(* IEC 61131-3 sources: Advanced_PLCs_Midterm_Project/Source_Code/Advanced_Midterm_PLC_Code/Dan_Thermostat_Code/Thermo_Code, 1 file *)

(* ---- HMI.plc ---- *)
PROGRAM PageDraw WITH Draw;
PROGRAM PageRefresh WITH Refresh;

	(***************************)
	(*                         *)
	(*     GLOBAL VARIABLES    *)
	(*                         *)
	(***************************)

VAR_GLOBAL

	{G:"Call stack"}
	giStackPtr : INT := -1;
	guiCallStack : ARRAY[ 0..9 ] OF UINT;

	{G:"Back buffer"}
	$giBackBufferCurr : INT := -1;
	$giBackBufferFirst : INT := -1;
	$giBackBufferLast : INT := -1;
	$guiBackBuffer : ARRAY[ 0..9 ] OF UINT;

	{G:"Sets"}
	$PagIndex : UINT;
	$PagNumber : UINT;
	$waitRefresh : BOOL;

	{G:"page1_vars"}
	fbpage1 : Drawpage1;
	fbRefrpage1 : Refrpage1;
	fbpage1String_1 : Static02 := (x:=58, y:=75, pFont:=?EWP2_8x16, bckCol:=12632256, pString:=?kStr00001, pVisVar:=1, format:=16#0020, bordPts:=0, selForeCol:=12632256, pRefrVar:=0, pSelVar:=0, numChars:=0);
	fbpage1String_4 : Static02 := (wHnd:=1, x:=54, y:=156, pFont:=?EWP2_8x16, bckCol:=12632256, pString:=?kStr00002, pVisVar:=1, format:=16#0020, bordPts:=0, selForeCol:=12632256, pRefrVar:=0, pSelVar:=0, numChars:=0);
	fbpage1Edit_3 : EditBox03 := (wHnd:=2, x1:=94, y1:=186, x2:=157, y2:=201, pFont:=?EWP2_8x16, bckCol:=32767, bordPts:=1, rw:=TRUE, pVar:=16#00201100, order:=2, pVisVar:=1, foreSelCol:=12632256, refr:=TRUE, type:=tyInt, format:=16#2100000C, pCanSel:=1, pEnumId:=0);
	fbpage1Edit_5 : EditBox03 := (wHnd:=3, x1:=91, y1:=100, x2:=154, y2:=115, pFont:=?EWP2_8x16, bckCol:=65535, bordPts:=1, rw:=TRUE, pVar:=16#00201000, order:=3, pVisVar:=1, foreSelCol:=12632256, refr:=TRUE, type:=tyInt, format:=16#2100000C, pCanSel:=1, pEnumId:=0);

	{G:"Back page manager"}
	fbBackPage : DrawBackPage;

END_VAR

	(***************************)
	(*                         *)
	(*        CONSTANTS        *)
	(*                         *)
	(***************************)

VAR_GLOBAL CONSTANT

	kStr00002 :STRING[18] := 'Relative Humidity';
	kStr00001 :STRING[19] := 'Temperature[deg F]';

END_VAR
VAR_GLOBAL CONSTANT

	{G:"Fonts"}
	EWP2_8x16_len : USINT := 8;
	EWP2_8x16_hei : USINT := 16;
	EWP2_8x16_offs : USINT := 0;
	EWP2_8x16 AT %MB1000.0 : ARRAY[ 0..2095 ] OF BYTE := 254,8,16,0,95,2,0,32,0,33,0,34,0,35,0,36,
				0,37,0,38,0,39,0,40,0,41,0,42,0,43,0,44,
				0,45,0,46,0,47,0,48,0,49,0,50,0,51,0,52,
				0,53,0,54,0,55,0,56,0,57,0,58,0,59,0,60,
				0,61,0,62,0,63,0,64,0,65,0,66,0,67,0,68,
				0,69,0,70,0,71,0,72,0,73,0,74,0,75,0,76,
				0,77,0,78,0,79,0,80,0,81,0,82,0,83,0,84,
				0,85,0,86,0,87,0,88,0,89,0,90,0,91,0,92,
				0,93,0,94,0,95,0,96,0,97,0,98,0,99,0,100,
				0,101,0,102,0,103,0,104,0,105,0,106,0,107,0,108,
				0,109,0,110,0,111,0,112,0,113,0,114,0,115,0,116,
				0,117,0,118,0,119,0,120,0,121,0,122,0,123,0,124,
				0,125,0,126,7(0),16,3(0),32,3(0),48,3(0),64,3(0),80,3(0),96,
				3(0),112,3(0),128,3(0),144,3(0),160,3(0),176,3(0),192,3(0),208,3(0),224,
				3(0),240,0,0,1,3(0),1,16,0,0,1,32,0,0,1,48,
				0,0,1,64,0,0,1,80,0,0,1,96,0,0,1,112,
				0,0,1,128,0,0,1,144,0,0,1,160,0,0,1,176,
				0,0,1,192,0,0,1,208,0,0,1,224,0,0,1,240,
				0,0,2,3(0),2,16,0,0,2,32,0,0,2,48,0,0,
				2,64,0,0,2,80,0,0,2,96,0,0,2,112,0,0,
				2,128,0,0,2,144,0,0,2,160,0,0,2,176,0,0,
				2,192,0,0,2,208,0,0,2,224,0,0,2,240,0,0,
				3,3(0),3,16,0,0,3,32,0,0,3,48,0,0,3,64,
				0,0,3,80,0,0,3,96,0,0,3,112,0,0,3,128,
				0,0,3,144,0,0,3,160,0,0,3,176,0,0,3,192,
				0,0,3,208,0,0,3,224,0,0,3,240,0,0,4,3(0),
				4,16,0,0,4,32,0,0,4,48,0,0,4,64,0,0,
				4,80,0,0,4,96,0,0,4,112,0,0,4,128,0,0,
				4,144,0,0,4,160,0,0,4,176,0,0,4,192,0,0,
				4,208,0,0,4,224,0,0,4,240,0,0,5,3(0),5,16,
				0,0,5,32,0,0,5,48,0,0,5,64,0,0,5,80,
				0,0,5,96,0,0,5,112,0,0,5,128,0,0,5,144,
				0,0,5,160,0,0,5,176,0,0,5,192,0,0,5,208,
				0,0,5,224,19(0),252,252,6(0),13,13,5(0),60,60,0,60,60,
				9(0),32,32,224,252,60,224,252,60,1,15,15,1,15,15,1,
				1,0,0,56,124,254,254,132,4,0,0,8,8,31,31,15,
				7,56,124,68,252,248,248,156,132,0,8,14,7,7,15,8,
				15,0,0,184,252,228,188,152,192,0,7,15,8,9,15,7,
				13,3(0),60,60,14(0),192,240,56,12,4,3(0),3,15,28,48,32,
				0,4,12,56,240,192,3(0),32,48,28,15,3,3(0),40,56,124,
				124,56,40,10(0),3(128),240,240,128,128,4(0),7,7,12(0),16,28,12,
				13(0),5(1),12(0),12,12,6(0),192,240,60,12,0,0,12,15,3,5(0),
				240,248,204,196,204,248,240,0,3,7,12,8,12,7,3,0,
				8,12,252,252,4(0),8,8,15,15,8,8,0,0,3(4),132,252,
				120,0,0,12,14,11,9,8,8,0,0,4,68,68,228,188,
				24,0,0,3(8),12,7,3,3(0),192,240,60,252,252,0,0,3,
				3,2,2,15,15,2,0,0,124,124,68,68,196,132,0,0,
				4(8),15,7,0,240,248,204,68,68,196,128,0,3,7,12,8,
				8,15,7,0,3(4),196,244,60,12,0,0,8,14,7,1,3(0),
				24,188,228,68,228,188,24,0,7,15,3(8),15,7,0,120,252,
				132,132,204,248,240,0,0,3(8),12,7,3,3(0),96,96,6(0),12,
				12,6(0),96,96,5(0),16,28,12,5(0),128,192,64,96,48,16,3(0),
				1,1,3,6,4,0,7(32),0,7(1),0,0,16,48,96,64,192,
				128,0,0,4,6,3,1,1,3(0),8,140,196,68,124,56,3(0),
				13,13,3(0),240,248,204,228,228,236,248,240,7,15,25,4(19),1,
				0,128,248,124,124,248,128,0,12,15,3,1,1,3,15,12,
				0,252,252,3(68),252,184,0,15,15,3(8),15,7,0,240,248,12,
				4,4,12,8,0,3,7,12,8,8,12,4,0,252,252,4,
				4,12,248,240,0,15,15,8,8,12,7,3,0,252,252,5(68),
				0,15,15,5(8),0,252,252,5(68),0,15,15,6(0),240,248,12,132,
				132,140,136,0,3,7,12,8,8,15,7,0,252,252,3(64),252,
				252,0,15,15,3(0),15,15,0,4,4,252,252,4,4,0,0,
				8,8,15,15,8,8,6(0),252,252,0,0,4(8),15,7,0,0,
				252,252,192,224,48,24,12,0,15,15,0,1,3,6,12,0,
				252,252,6(0),15,15,5(8),0,252,252,120,96,120,252,252,0,15,
				15,3(0),15,15,0,252,252,120,224,128,252,252,0,15,15,0,
				1,7,15,15,0,240,248,12,4,12,248,240,0,3,7,12,
				8,12,7,3,0,252,252,3(68),124,56,0,15,15,6(0),240,248,
				12,4,12,248,240,0,3,7,12,24,60,39,35,0,252,252,
				68,196,196,124,56,0,15,15,0,0,3,7,12,0,56,124,
				68,196,132,140,8,0,4,12,3(8),15,7,3(4),252,252,3(4),3(0),
				15,15,4(0),252,252,3(0),252,252,0,7,15,3(8),15,7,12,124,
				240,128,128,240,124,12,0,0,7,15,15,7,0,0,252,252,
				128,224,224,128,252,252,3,15,15,3,3,15,15,3,4,28,
				56,224,224,56,28,4,8,14,7,1,1,7,14,8,4,28,
				56,224,224,56,28,4,3(0),15,15,4(0),4,4,132,228,116,28,
				12,0,12,14,11,9,3(8),3(0),252,252,4,4,4(0),63,63,32,
				32,0,0,12,60,240,192,7(0),3,15,12,0,0,4,4,252,
				252,4(0),32,32,63,63,4(0),64,112,56,12,12,56,112,16(0),8(64),
				3(0),4,12,8,11(0),64,96,3(32),224,192,0,6,15,9,9,13,
				15,15,0,252,252,96,32,96,192,128,0,15,15,12,8,12,
				7,3,0,128,192,96,4(32),0,3,7,12,4(8),0,128,192,96,
				32,96,252,252,0,3,7,12,8,12,15,15,0,128,192,96,
				32,96,192,128,0,3,7,13,4(9),0,32,32,248,252,3(36),3(0),
				15,15,4(0),192,224,32,32,224,224,32,0,61,127,74,74,75,
				121,48,0,252,252,96,32,32,224,192,0,15,15,3(0),15,15,
				0,0,32,32,228,228,6(0),15,15,4(0),32,32,228,228,3(0),3(64),
				127,63,3(0),252,252,128,192,96,32,0,0,15,15,1,3,6,
				12,8,0,4,4,252,252,6(0),15,15,8,8,0,224,224,32,
				224,224,32,224,192,15,15,0,15,15,0,15,15,0,224,224,
				96,32,32,224,192,0,15,15,3(0),15,15,0,192,224,3(32),224,
				192,0,7,15,3(8),15,7,0,224,224,96,32,96,192,128,0,
				127,127,12,8,12,7,3,0,128,192,96,32,96,224,224,0,
				3,7,12,8,12,127,127,0,0,224,224,96,3(32),0,0,15,
				15,5(0),192,224,5(32),0,8,4(9),15,6,0,0,32,248,248,32,
				32,4(0),7,15,3(8),0,224,224,3(0),224,224,0,7,15,8,8,
				12,15,15,32,224,192,0,0,192,224,32,0,1,7,14,14,
				7,1,0,224,224,0,128,128,0,224,224,3,15,15,3,3,
				15,15,3,0,32,96,192,128,192,96,32,0,8,12,7,3,
				7,12,8,32,224,192,0,0,192,224,32,64,64,103,63,31,
				7,3(0),3(32),160,224,96,32,0,8,12,15,11,3(8),0,0,128,
				248,124,4,5(0),31,63,32,5(0),252,252,6(0),63,63,6(0),4,124,
				248,128,4(0),32,63,31,3(0),4(128),0,0,128,1,1,0,0,4(1);

	{G:"Keys"}
	kKEY_Enter : USINT := 13;
	kKEY_Esc : USINT := 27;
	kKEY_Del : USINT := 127;
	kKEY_Left : USINT := 8;
	kKEY_Right : USINT := 12;
	kKEY_ArrowUp : USINT := 11;
	kKEY_ArrowDw : USINT := 10;
	kKEY_Back : USINT := 4;
	kKEY_Tab : USINT := 9;
	kKEY_Shift : USINT := 6;
	kKEY_Caps : USINT := 5;
	kKEY_Confirm : USINT := 14;
	kKEY_VK_F1 : USINT := 30;
	kKEY_VK_F2 : USINT := 31;
	kKEY_VK_F3 : USINT := 32;
	kKEY_VK_F4 : USINT := 33;
	kKEY_VK_F5 : USINT := 34;
	kKEY_VK_F6 : USINT := 35;
	kKEY_VK_F7 : USINT := 36;
	kKEY_VK_F8 : USINT := 37;
	kKEY_VK_F9 : USINT := 38;
	kKEY_VK_F10 : USINT := 39;

	{G:"Data types"}
	tyUndefined : USINT := 19;
	tyBool : USINT := 1;
	tySInt : USINT := 2;
	tyInt : USINT := 5;
	tyDInt : USINT := 9;
	tyLInt : USINT := 12;
	tyUSInt : USINT := 3;
	tyUInt : USINT := 6;
	tyUDInt : USINT := 10;
	tyULInt : USINT := 13;
	tyReal : USINT := 15;
	tyLReal : USINT := 16;
	tyByte : USINT := 4;
	tyWord : USINT := 7;
	tyDWord : USINT := 11;
	tyLWord : USINT := 14;
	tyString : USINT := 17;

	{G:"Messages"}
	kWM_NULL : UINT := 0;
	kWM_KEY : UINT := 1;
	kWM_MSG : UINT := 2;
	kWM_SELECT : UINT := 3;
	kWM_PUSH : UINT := 4;
	kEV_WM_TEXTSELECT : UINT := 5;
	kEV_WM_OPENPAGE : UINT := 6;
	kEV_WM_CLOSEPAGE : UINT := 7;
	kEV_WM_CHANGESETPAGE : UINT := 8;

	{G:"Access modes"}
	kACS_IDLE : USINT := 0;
	kACS_INIT : USINT := 1;
	kACS_PRINT : USINT := 2;
	kACS_SELECT : USINT := 3;
	kACS_MODIFY : USINT := 4;
	kACS_DELETE : USINT := 5;
	kACS_QUERY : USINT := 6;
	kACS_BCKQUERY : USINT := 7;
	kACS_CLOSE : USINT := 8;
	kACS_OPEN : USINT := 9;

	{G:"Parameters and device"}
	kCOMM_PROTO_ID_LOCAL : USINT := 1;
	kCOMM_PROTO_ID_MODBUS_RTU : USINT := 2;
	kCOMM_PROTO_ID_MODBUS_TCP : USINT := 3;
	kCOMM_PROTO_ID_CANOPEN : USINT := 4;

	{G:"Button types"}
	kBTN_TYPE_NORMAL : USINT := 0;
	kBTN_TYPE_TOGGLE : USINT := 1;

	{G:"Resources"}
	kLangBaseLanguage : UDINT := 0;

	(*** Enumeratives: ***)

	{G:"Parameters"}
	kPAR_MSG_NOTFOUND : UINT := 103;
	kPAR_MSG_SYSERR : UINT := 106;
	kPAR_ERR_OK : UINT := 0;
	kPAR_ERR_NOTFOUND : UINT := 1;
	kPAR_ERR_INVTYPE : UINT := 3;

END_VAR

	(***************************)
	(*                         *)
	(*        PROGRAMS         *)
	(*                         *)
	(***************************)

PROGRAM PageDraw

	VAR
	res : USINT;
	END_VAR

	{CODE:ST}
	(* Locking the video *)
	res := Video_Lock( res );

	(* The resource bitmaps color depth is supported... *)
	res := Video_SetUseBitmapsColorDepth( TRUE );

	(* INIT HMI ENVIRONMENT *)
	res := Video_InitHMI_ZOrder( TRUE );

	(* Switching on the LCD *)
	res := Video_Switch( TRUE );

	(* Initializing the length of the call stack *)
	giStackPtr := 0;

	(* Initializing the back circular buffer indexes *)
	$giBackBufferCurr := -1;
	$giBackBufferFirst := -1;
	$giBackBufferLast := -1;

	(* Declaring the code of the keys for driving the editing mode *)
	res := Video_SetEditKey( 0, kKEY_Enter );
	res := Video_SetEditKey( 1, kKEY_Esc );
	res := Video_SetEditKey( 2, kKEY_Del );
	res := Video_SetEditKey( 3, kKEY_Left );
	res := Video_SetEditKey( 4, kKEY_Right );
	res := Video_SetEditKey( 5, kKEY_ArrowUp );
	res := Video_SetEditKey( 6, kKEY_ArrowDw );
	res := Video_SetEditKey( 7, kKEY_Back );
	res := Video_SetEditKey( 8, kKEY_Tab );
	res := Video_SetEditKey( 9, kKEY_Shift );
	res := Video_SetEditKey( 10, kKEY_Caps );
	res := Video_SetEditKey( 11, kKEY_Confirm );

	(* *** DECLARING THE RESOURCES *** *)
	res := Video_LoadLanguage( 0, 0 );

	(* Declaring the imported fonts *)
	res := Video_AddFontUnicode( ?EWP2_8x16, EWP2_8x16_len, EWP2_8x16_hei );

	(* Declaring the system attributes of windows *)
	res := Video_SetWndSysProps( ?EWP2_8x16, 12632256, 0 );

	(* *** INITIALIZING THE OBJECTS OF PAGE 'page1' *** *)

	(* Init the set elements *)
	guiCallStack[ giStackPtr ] := 0;
	WHILE TRUE DO
		CASE guiCallStack[ giStackPtr ] OF

			0:
				fbpage1();

		END_CASE;

	END_WHILE;

END_PROGRAM

PROGRAM PageRefresh

VAR
res : USINT;
END_VAR

	{CODE:ST}
	(* Wait for the PageDraw to start *)
	WHILE giStackPtr < 0 DO
		res := Video_Sleep(50);
	END_WHILE;

	WHILE TRUE DO
		CASE guiCallStack[ giStackPtr ] OF

			0:
				fbRefrpage1();

		END_CASE;

		res := Video_Sleep( 50 );

	END_WHILE;

END_PROGRAM

	(***************************)
	(*                         *)
	(*  ALARM PAGE F. BLOCKS   *)
	(*                         *)
	(***************************)

FUNCTION_BLOCK DrawBackPage

	VAR_INPUT
		IsOpening : BOOL;
		CurrPageId : UINT;
	END_VAR
	VAR_OUTPUT
		BackPageId : UINT;
	END_VAR
	VAR_EXTERNAL
		$giBackBufferCurr : INT;
		$giBackBufferFirst : INT;
		$giBackBufferLast : INT;
		$guiBackBuffer : ARRAY[ 0..9 ] OF UINT;
	END_VAR
	{CODE:ST}

	IF IsOpening THEN

		(* Entering page *)

		(* Save this page's ID into circular back buffer *)
		$giBackBufferCurr := $giBackBufferCurr + 1;
		IF $giBackBufferCurr >= 10 THEN
			$giBackBufferCurr := 0;
		END_IF;
		$guiBackBuffer[ $giBackBufferCurr ] := CurrPageId;
		IF $giBackBufferFirst = -1 THEN
			$giBackBufferFirst := 0;
		ELSIF $giBackBufferCurr = $giBackBufferFirst AND $giBackBufferFirst <> $giBackBufferLast THEN
			$giBackBufferFirst := $giBackBufferFirst + 1;
			IF $giBackBufferFirst = 10 THEN
				$giBackBufferFirst := 0;
			END_IF;
		END_IF;

		(* Set last page's ID *)
		IF $giBackBufferCurr = $giBackBufferFirst THEN
			$giBackBufferLast := -1;
		ELSIF $giBackBufferCurr = 0 AND $giBackBufferFirst <> 9 THEN
			$giBackBufferLast := 9;
		ELSIF $giBackBufferCurr <> $giBackBufferFirst THEN
			$giBackBufferLast := $giBackBufferCurr - 1;
		ELSE
			$giBackBufferLast := -1;
		END_IF;
		IF $giBackBufferLast <> -1 THEN
			BackPageId := $guiBackBuffer[$giBackBufferLast];
		ELSE
			BackPageId := 16#FFFF;
		END_IF;

	ELSE

		(* Closing page *)
		$giBackBufferCurr := $giBackBufferCurr - 1;
		IF $giBackBufferCurr < 0 THEN
			$giBackBufferCurr := 9;
		END_IF;
		$giBackBufferCurr := $giBackBufferCurr - 1;
		IF $giBackBufferCurr < 0 THEN
			$giBackBufferCurr := 9;
		END_IF;

	END_IF;

	END_FUNCTION_BLOCK

	(***********************************)
	(*                                 *)
	(* EXPRESSIONS RESOLVER F. BLOCKS  *)
	(*                                 *)
	(***********************************)

	(***************************)
	(*                         *)
	(* PAGE-DRAWING F. BLOCKS  *)
	(*                         *)
	(***************************)

FUNCTION_BLOCK Drawpage1

	VAR_OUTPUT
	uiOutVar : UINT;
	END_VAR

	VAR_EXTERNAL
	guiCallStack : ARRAY[ 0..9 ] OF UINT;
	giStackPtr : INT;
	fbBackPage : DrawBackPage;
	fbpage1String_1 : Static02;
	fbpage1String_4 : Static02;
	fbpage1Edit_3 : EditBox03;
	fbpage1Edit_5 : EditBox03;
	$waitRefresh : BOOL;
	END_VAR

	VAR
	res : USINT;
	bStatRedrw : BOOL;
	bMapsReset : BOOL;
	iNextSel : INT;
	$Set_IndexVisEl : UINT;
	$Set_CycleRefresh : UINT;
	$Set_PtrBoolVis : @BOOL;
	$Set_VisEl : BOOL;
	$Set_IndexPageInSet : UINT;
	$Set_ForcePageReload : BOOL;
	$Set_NextPage : BOOL;
	$Set_PrevPage : BOOL;
	$Set_LocalSetPagNumber: UINT;
	$Set_NumVisEl: UINT;
	$Set_LastFirstEl: INT;
	udiev : UDINT;
	ev : UINT;
	key : USINT;
	x1 : UINT;
	y1 : UINT;
	x2 : UINT;
	y2 : UINT;
	wParam : UINT;
	END_VAR

	{CODE:ST}

	(* Writing this page's ID to the top of the callstack *)
	guiCallStack[ giStackPtr ] := 16#00;

	(* Manage back page index for opening page *)
	fbBackPage.IsOpening := TRUE;
	fbBackPage.CurrPageId := 16#00;
	fbBackPage();

	(* Flag of waiting for refresh task *)
	$waitRefresh := TRUE;

	(* Resetting the object map *)
	res := Video_ResetMaps( 16#00 );

	(* Setting flags: this page is to be drawn *)
	bStatRedrw := TRUE;
	bMapsReset := TRUE;

	(* The area to be cleared is the area of the entire page *)
	x1:= 0;
	y1:= 0;
	x2:= 239;
	y2:= 319;

	(* Unlocking the video *)
	res := Video_Unlock( res );

	WHILE TRUE DO

		(* Locking the video *)
		res := Video_Lock( res );

		(* Initializing the page *)
		res := Video_InitPage( 0, 0, 239, 319, ?' ', 16#0003 );

		(* Setting the page colors *)
		res := Video_SetPageColors( 0, 12632256 );

		IF bStatRedrw THEN

			(* *** CLEARING PAGE AREA *** *)
			res := Video_ClrRect( x1, y1, x2, y2 );

		END_IF;

		IF bMapsReset THEN

			(* Resetting all maps *)
			res := Video_ResetMaps( 16#FF );

			(* *** DRAW PAGE CONTROLS *** *)

			(* *** PAGE SECTION *** *)

			(* *** DRAW CONTROLS *** *)
			fbpage1String_1.accMode := kACS_INIT;
			fbpage1String_1();
			fbpage1String_1.accMode := kACS_PRINT;
			fbpage1Edit_3.accMode := kACS_INIT;
			fbpage1Edit_3();
			fbpage1Edit_3.accMode := kACS_PRINT;
			fbpage1String_4.accMode := kACS_INIT;
			fbpage1String_4();
			fbpage1String_4.accMode := kACS_PRINT;
			fbpage1Edit_5.accMode := kACS_INIT;
			fbpage1Edit_5();
			fbpage1Edit_5.accMode := kACS_PRINT;

		END_IF;

		(* Unlocking the video *)
		res := Video_Unlock( res );

		(* Reset the flags for page redraw request *)
		bStatRedrw := FALSE;
		bMapsReset := FALSE;

		(* *** EVENTS HANDLING *** *)
		WHILE NOT bStatRedrw DO

			(* the drawing task wait the refreshing task *)
			IF $waitRefresh THEN
				res := Video_Sleep( 50 );
			ELSE

				(* Retrieving events *)
				udiev := Video_GetEvent( res );
				(* Extracting the event code *)
				ev := TO_UINT(udiev);

				CASE ev OF

				(* Key-related events handling: *)
				kWM_KEY:

					key := TO_USINT(SHR(udiev, 16));

				(* Selecting a control: *)
				kWM_SELECT:

					(* Extracting the index of the edit box clicked *)
					iNextSel := TO_INT(SHR(udiev, 16));

					CASE iNextSel OF

						2,3:
							REPEAT

							(* Entering the edit mode *)
							res := Video_EnterEdit( TO_UINT( iNextSel ) );

							IF res = kKEY_ArrowUp THEN

								iNextSel := TO_INT( Video_NextEdit( TRUE ) );
								IF iNextSel > -1 THEN
									res := Video_SendEvent( kWM_SELECT, TO_UINT(iNextSel) );
								END_IF;

							ELSIF res = kKEY_ArrowDw THEN

								iNextSel := TO_INT( Video_PrevEdit( TRUE ) );
								IF iNextSel > -1 THEN
									res := Video_SendEvent( kWM_SELECT, TO_UINT(iNextSel) );
								END_IF;

							END_IF;

							UNTIL res <> kKEY_Confirm
							END_REPEAT;

							IF res <> 255 THEN
								(* The area to be cleared is the area of the entire screen (without system bar)*)
								x1:= 0;
								y1:= 0;
								x2:= 239;
								y2:= 319;
								bMapsReset := TRUE;
								bStatRedrw := TRUE;
							END_IF;

					END_CASE;

					END_CASE;
				END_IF;

			END_WHILE;

		END_WHILE;

	END_FUNCTION_BLOCK

	(***************************)
	(*                         *)
	(* REFRESHING FUN. BLOCKS  *)
	(*                         *)
	(***************************)

FUNCTION_BLOCK Refrpage1

	VAR_EXTERNAL
	guiCallStack : ARRAY[ 0..9 ] OF UINT;
	giStackPtr : INT;
	fbpage1String_1 : Static02;
	fbpage1String_4 : Static02;
	fbpage1Edit_3 : EditBox03;
	fbpage1Edit_5 : EditBox03;
	$waitRefresh : BOOL;
	END_VAR

	VAR
	res : USINT;
	pagID : UINT;
	n : USINT;
	iSP : INT;
	pDC : UDINT;
	rx1 : UINT;
	ry1 : UINT;
	rx2 : UINT;
	ry2 : UINT;
	END_VAR

	{CODE:ST}

	REPEAT

		(* Locking the video *)
		res := Video_Lock( res );

		(* Testing if page has changed *)
		pagID := guiCallStack[ giStackPtr ];

		IF pagID = 16#00 THEN

			(* the refresh task is arrived *)
			$waitRefresh := FALSE;

			(* *** REFRESH PAGE CONTROLS *** *)

			(* Update refresh flags for page controls *)
			res := Video_UpdatePageControls( TRUE );

			(* *** REFRESHING BACKGROUND ITEMS *** *)
			(* Cursor across the call stack *)
			iSP := giStackPtr;

			(* *** REFRESHING PARENT BACKGROUND ITEMS *** *)

		END_IF;

		(* Unlocking the video *)
		res := Video_Unlock( res );

		(* Suspending the task *)
		res := Video_Sleep( 50 );

	UNTIL pagID <> 16#00
	END_REPEAT;

END_FUNCTION_BLOCK

	(***************************)
	(*                         *)
	(* PARAMETER  FUN. BLOCKS  *)
	(*                         *)
	(***************************)

	(*****************************)
	(*                           *)
	(*     ID RES. CONSTANTS     *)
	(*                           *)
	(*****************************)

(************************************************************************)
(*                                                                      *)
(*	Description: Definition of target variables and functions       *)
(*                                                                      *)
(************************************************************************)

(************************************************************************)
(*                         									                            *)
(*   GLOBAL VARIABLES                                                   *)
(*                                                                      *)
(************************************************************************)

(************************************************************************)
(*                        		  *)
(*   CUSTOM EMBEDDED FUNCTIONS    *)
(*                         		  *)
(************************************************************************)
FUNCTION Video_GetPixelColor : UDINT

	VAR_INPUT
	xPos : UINT;
	yPos : UINT;
	END_VAR

	{CODE:EMBEDDED}

END_FUNCTION

(* !!!!!! IMPORTANT: CONTENTS OF THIS MODULE SHOULD BE KEPT ALIGNED WITH AlHMIIec.h !!!!!! *)

(************************************************************************)
(*                         *)
(*   EMBEDDED FUNCTIONS    *)
(*                         *)
(************************************************************************)
FUNCTION Video_InitHMI_ZOrder : BOOL

	VAR_INPUT
	dmy : BOOL;
	END_VAR

	{CODE:EMBEDDED}

END_FUNCTION

FUNCTION Video_LCDContrast : BOOL

	VAR_INPUT
	more : BOOL;
	END_VAR

	{CODE:EMBEDDED}

END_FUNCTION

FUNCTION Video_Switch : USINT

	VAR_INPUT
	on : USINT;
	END_VAR

	{CODE:EMBEDDED}

END_FUNCTION

FUNCTION Video_DrawFrames : USINT

	VAR_INPUT
	left : UINT;
	top : UINT;
	right : UINT;
	bottom : UINT;
	colBack : UDINT;
	fBar : USINT;
	pTitle : UDINT;
	fResStr : BOOL;
	fSysBtn : USINT;
	style : USINT;
	END_VAR

	{CODE:EMBEDDED}

END_FUNCTION

FUNCTION Video_InitPage : USINT

	VAR_INPUT
	x1 : UINT;
	y1 : UINT;
	x2 : UINT;
	y2 : UINT;
	pTitle : UDINT;
	wData : UINT;
	END_VAR

	{CODE:EMBEDDED}

END_FUNCTION

FUNCTION Video_ClrRect : USINT

	VAR_INPUT
	x1 : UINT;
	y1 : UINT;
	x2 : UINT;
	y2 : UINT;
	END_VAR

	{CODE:EMBEDDED}

END_FUNCTION

FUNCTION Video_ClrScreen : BOOL

	VAR_INPUT
	dummy : USINT;
	END_VAR

	{CODE:EMBEDDED}

END_FUNCTION

FUNCTION Video_SaveRect : USINT

	VAR_INPUT
	x1 : UINT;
	y1 : UINT;
	x2 : UINT;
	y2 : UINT;
	END_VAR

	{CODE:EMBEDDED}

END_FUNCTION

FUNCTION Video_WriteFromBuff : USINT

	VAR_INPUT
	x1 : UINT;
	y1 : UINT;
	x2 : UINT;
	y2 : UINT;
	END_VAR

	{CODE:EMBEDDED}

END_FUNCTION

FUNCTION Video_SetPageColors : USINT

	VAR_INPUT
	colFore : UDINT;
	colBack : UDINT;
	END_VAR

	{CODE:EMBEDDED}

END_FUNCTION

FUNCTION Video_SetWndSysProps : USINT

	VAR_INPUT
	pFont	: UDINT;
	colFore : UDINT;
	colBack : UDINT;
	END_VAR

	{CODE:EMBEDDED}

END_FUNCTION

FUNCTION Video_SetEditKey : USINT

	VAR_INPUT
	id : USINT;
	code : USINT;
	END_VAR

	{CODE:EMBEDDED}

END_FUNCTION

FUNCTION Video_AddFont : USINT

	VAR_INPUT
	pFont : UDINT;
	charLen : USINT;
	charHei : USINT;
	offs : USINT;
	END_VAR

	{CODE:EMBEDDED}

END_FUNCTION

FUNCTION Video_AddFontUnicode : USINT

	VAR_INPUT
	pFont : UDINT;
	charLen : UINT;
	charHei : USINT;
	END_VAR

	{CODE:EMBEDDED}

END_FUNCTION

FUNCTION Video_SetFont : USINT

	VAR_INPUT
	fontPtr : UDINT;
	END_VAR

	{CODE:EMBEDDED}

END_FUNCTION

FUNCTION Video_LoadExternalFont : UDINT
	{ DE:"Load an external font from PLK file on disk" }
	VAR_INPUT
	filename : STRING;
	END_VAR

	{CODE:EMBEDDED}
END_FUNCTION

FUNCTION Video_SetColors : USINT

	VAR_INPUT
	colForeTxt : UDINT;
	colBackTxt : UDINT;
	colForeSel : UDINT;
	colBackSel : UDINT;
	END_VAR

	{CODE:EMBEDDED}

END_FUNCTION

FUNCTION Video_Line : USINT

	VAR_INPUT
	x1 : UINT;
	y1 : UINT;
	x2 : UINT;
	y2 : UINT;
	pts : USINT;
	color : UDINT;
	END_VAR

	{CODE:EMBEDDED}

END_FUNCTION

FUNCTION Video_Rectangle : USINT

	VAR_INPUT
	x1 : UINT;
	y1 : UINT;
	x2 : UINT;
	y2 : UINT;
	pts : USINT;
	transp : USINT;
	bordCol : UDINT;
	fillCol : UDINT;
	END_VAR

	{CODE:EMBEDDED}

END_FUNCTION

FUNCTION Video_PrintStr : USINT

	VAR_INPUT
	str : STRING;
	x : UINT;
	y : UINT;
	END_VAR

	{CODE:EMBEDDED}

END_FUNCTION

FUNCTION Video_PrintResStr : USINT

	VAR_INPUT
	idRes : UINT;
	x : UINT;
	y : UINT;
	END_VAR

	{CODE:EMBEDDED}

END_FUNCTION

FUNCTION Video_PrintResStrByName : USINT

	VAR_INPUT
	resName : STRING;
	x : UINT;
	y : UINT;
	END_VAR

	{CODE:EMBEDDED}

END_FUNCTION

FUNCTION Video_PrintNChar : USINT

	VAR_INPUT
	str : STRING;
	accMode : USINT;
	x : UINT;
	y : UINT;
	nChar : USINT;
	format : UDINT;
	END_VAR

	{CODE:EMBEDDED}

END_FUNCTION

FUNCTION Video_PrintBitmap : USINT

	VAR_INPUT
		ptrBmp : UDINT;
		x : UINT;
		y : UINT;
	END_VAR

	{CODE:EMBEDDED}

END_FUNCTION

FUNCTION Video_DelBitmap : USINT

	VAR_INPUT
		ptrBmp : UDINT;
		x : UINT;
		y : UINT;
	END_VAR

	{CODE:EMBEDDED}

END_FUNCTION

FUNCTION Video_DrawBorder : USINT

	VAR_INPUT
		style : USINT;
		x1 : UINT;
		y1 : UINT;
		x2 : UINT;
		y2 : UINT;
		pts : USINT;
		color : UDINT;
	END_VAR

	{CODE:EMBEDDED}

END_FUNCTION

FUNCTION Video_DelBorder : USINT

	VAR_INPUT
		style : USINT;
		x1 : UINT;
		y1 : UINT;
		x2 : UINT;
		y2 : UINT;
		pts : USINT;
	END_VAR

	{CODE:EMBEDDED}

END_FUNCTION

FUNCTION Video_SendEvent : USINT

	VAR_INPUT
	msgID : UINT;
	wParam : UINT;
	END_VAR

	{CODE:EMBEDDED}

END_FUNCTION

FUNCTION Video_GetEvent : UDINT

	VAR_INPUT
	dmy : USINT;
	END_VAR

	{CODE:EMBEDDED}

END_FUNCTION

FUNCTION Video_EnterEdit : USINT

	VAR_INPUT
	wHnd : UINT;
	END_VAR

	{CODE:EMBEDDED}

END_FUNCTION

FUNCTION Video_EnterEditSel : USINT

	VAR_INPUT
	wHnd : UINT;
	onlySelect : BOOL;
	END_VAR

	{CODE:EMBEDDED}

END_FUNCTION

FUNCTION Video_NextEdit : UINT

	VAR_INPUT
	fRWOnly : USINT;
	END_VAR

	{CODE:EMBEDDED}

END_FUNCTION

FUNCTION Video_FirstLastEdit : INT

	VAR_INPUT
	fRWOnly : BOOL;
	last : BOOL;
	END_VAR

	{CODE:EMBEDDED}

END_FUNCTION

FUNCTION Video_PrevEdit : UINT

	VAR_INPUT
	fRWOnly : USINT;
	END_VAR

	{CODE:EMBEDDED}

END_FUNCTION

FUNCTION Video_PushButton : USINT

	VAR_INPUT
	wHnd : UINT;
	END_VAR

	{CODE:EMBEDDED}

END_FUNCTION

FUNCTION Video_Lock : USINT

	VAR_INPUT
	res : USINT;
	END_VAR

	{CODE:EMBEDDED}

END_FUNCTION

FUNCTION Video_Unlock : USINT

	VAR_INPUT
	res : USINT;
	END_VAR

	{CODE:EMBEDDED}

END_FUNCTION

FUNCTION Video_Sleep : USINT

	VAR_INPUT
	msec : UINT;
	END_VAR

	{CODE:EMBEDDED}

END_FUNCTION

FUNCTION Video_ResetMaps : USINT

	VAR_INPUT
	res : USINT;
	END_VAR

	{CODE:EMBEDDED}

END_FUNCTION

FUNCTION Video_LoadLanguage : USINT

	VAR_INPUT
	pResStrings : UDINT;	{DE:"Pointer to resource strings of active language"}
	pEnums : UDINT;			{DE:"Pointer to enumerated types of active language"}
	END_VAR

	{CODE:EMBEDDED}

END_FUNCTION

FUNCTION Video_EvNotify : USINT

	VAR_INPUT
	evId : UINT;	{DE:"Event ID"}
	data0 : UDINT;			{DE:"Event custom data0"}
	data1 : UDINT;			{DE:"Event custom data1"}
	END_VAR

	{CODE:EMBEDDED}

END_FUNCTION

FUNCTION Video_InitBmpTreeRefresh : UDINT

	VAR_INPUT
	x1 : UINT; {DE:"X-coordinate of the upper-left corner"}
	y1 : UINT; {DE:"Y-coordinate of the upper-left corner"}
	x2 : UINT; {DE:"X-coordinate of the lower-right corner"}
	y2 : UINT; {DE:"Y-coordinate of the lower-right corner"}
	END_VAR

	{CODE:EMBEDDED}

END_FUNCTION

FUNCTION Video_EndBmpTreeRefresh : USINT

	VAR_INPUT
	pDC : UDINT; {DE:"Pointer to the device context"}
	x1  : UINT;  {DE:"X-coordinate of the upper-left corner"}
	y1  : UINT;  {DE:"Y-coordinate of the upper-left corner"}
	x2  : UINT;  {DE:"X-coordinate of the lower-right corner"}
	y2  : UINT;  {DE:"Y-coordinate of the lower-right corner"}
	END_VAR

	{CODE:EMBEDDED}

END_FUNCTION

FUNCTION Video_ForceRefresh : BOOL

	VAR_INPUT
	dummy : USINT;
	END_VAR

	{CODE:EMBEDDED}

END_FUNCTION

FUNCTION Video_IsInEdit : BOOL

	VAR_INPUT
	dummy : USINT;
	END_VAR

	{CODE:EMBEDDED}

END_FUNCTION

FUNCTION Video_SetStrAndEnumsOnTgt : BOOL
	{ DE:"Set the resource on target" }
	VAR_INPUT
	enable : BOOL;	{ DE:"Enable the resource on the target " }
	END_VAR
	{ CODE:EMBEDDED }
END_FUNCTION

FUNCTION Video_SetBitmapsOnTgt: BOOL
    { DE:"Set the bitmaps on target" }
    VAR_INPUT
    enable : BOOL;    { DE:"Enable the bitmaps on the target " }
    END_VAR
    { CODE:EMBEDDED }
END_FUNCTION

FUNCTION Video_AddExternalBmp: BOOL
	{ DE:"Add a bitmap in code as external bitmap" }
    VAR_INPUT
	name : STRING; { DE:"Name of the bitmap" }
    addr : UDINT;    { DE:"Address of the bitmap" }
    END_VAR
    { CODE:EMBEDDED }
END_FUNCTION

FUNCTION Video_GetParamBckgnd : UINT

	VAR_INPUT
	idxDevice 	: USINT;	{DE:"index of device"}
	idxParam 	: UINT; 	{DE:"index of param"}
	subIdxParam : USINT; 	{DE:"sub index of param"}

	pVal : UDINT;			{DE:"Pointer to value of parameter"}
	type : USINT; 			{DE:"Data type of the associated variable"}
	aux  : UDINT;			{DE:"Reserved for future use"}
	END_VAR

	{CODE:EMBEDDED}

END_FUNCTION

FUNCTION Video_SetParam : UINT

	VAR_INPUT
	idxDevice 	: USINT;	{DE:"index of device"}
	idxParam 	: UINT; 	{DE:"index of param"}
	subIdxParam : USINT; 	{DE:"sub index of param"}

	pVal : UDINT;			{DE:"Pointer to value of parameter"}
	type : USINT; 			{DE:"Data type of the associated variable"}
	END_VAR

	{CODE:EMBEDDED}

END_FUNCTION

FUNCTION Video_GetParam : UINT

	VAR_INPUT
	idxDevice 	: USINT;	{DE:"index of device"}
	idxParam 	: UINT; 	{DE:"index of param"}
	subIdxParam : USINT; 	{DE:"sub index of param"}

	pVal : UDINT;			{DE:"Pointer to value of parameter"}
	type : USINT; 			{DE:"Data type of the associated variable"}
	END_VAR

	{CODE:EMBEDDED}

END_FUNCTION

(*FUNCTION sysHmi_Message : BOOL
	{ DE:"Open a Message window on display" }
	VAR_INPUT
	    id	:  USINT; { DE:"User Message window ID [1..99]" }
	END_VAR
	{CODE:EMBEDDED}
END_FUNCTION*)

FUNCTION Video_DrawStaticControls : BOOL

	VAR_INPUT
	staticMode	: BOOL;		{DE:"Activate or deactivate static control drawing"}
	END_VAR

	{CODE:EMBEDDED}

END_FUNCTION

FUNCTION Video_SSaver_IsActive : BOOL
	VAR_INPUT
	dmy : USINT;
	END_VAR

	{CODE:EMBEDDED}
END_FUNCTION

FUNCTION Video_SSaver_SetTimeout : BOOL
	VAR_INPUT
	seconds : UINT;
	END_VAR

	{CODE:EMBEDDED}
END_FUNCTION

FUNCTION Video_SSaver_GetTimeout : UINT
	VAR_INPUT
	dmy : USINT;
	END_VAR

	{CODE:EMBEDDED}
END_FUNCTION

FUNCTION Video_SSaver_GetRemTime : UINT
	VAR_INPUT
	dmy : USINT;
	END_VAR

	{CODE:EMBEDDED}
END_FUNCTION

FUNCTION Video_SetUseBitmapsColorDepth : BOOL
	VAR_INPUT
	useColorDepth : BOOL;
	END_VAR

	{CODE:EMBEDDED}
END_FUNCTION

FUNCTION Video_UpdatePageControls : BOOL
	VAR_INPUT
		dmy : BOOL;
	END_VAR

	{CODE:EMBEDDED}
END_FUNCTION

FUNCTION Video_LoadLanguageOffsetIndex : USINT
    VAR_INPUT
    pResStrings : UDINT;             {DE:"Pointer to resource strings of active language"}
    pEnums : UDINT;                  {DE:"Pointer to enumerated types of active language"}
    pResStringsOffsetIndex : UDINT;  {DE:"Pointer to resource strings map index of active language"}
    pEnumsOffsetIndex : UDINT;       {DE:"Pointer to resource enums map index of active language"}
    END_VAR

{CODE:EMBEDDED}
END_FUNCTION

	(***************************)
	(*                         *)
	(*  EMBEDDED FUN. BLOCKS   *)
	(*                         *)
	(***************************)

FUNCTION_BLOCK Video_GetPageColors

	VAR_OUTPUT
	color : UDINT;	{DE:"Actual page foreground color"}
	back : UDINT;	{DE:"Actual page background color"}
	END_VAR

	{CODE:EMBEDDED}

END_FUNCTION_BLOCK

	(***************************)
	(*                         *)
	(*         OBJECTS         *)
	(*                         *)
	(***************************)

FUNCTION_BLOCK Static01

	VAR_INPUT
	wHnd : UINT; {DE:"Object handle"}
	x : UINT; {DE:"X-coordinate of the upper-left corner"}
	y : UINT; {DE:"Y-coordinate of the upper-left corner"}
	accMode : USINT; {DE:"Access mode"}
	fResStr : BOOL; {DE:"Flag for resource strings"}
	pString : UDINT; {DE:"Address of the string"}
	pFont : UDINT; {DE:"Address of the font"}
	foreCol : UDINT; {DE:"Foreground color"}
	bckCol : UDINT; {DE:"Background color"}
	pVisVar : UDINT; {DE:"Address of the visibility flag"}
	format : UINT; {DE:"Alignment of static"}
	style : USINT; {DE:"Appearence"}
	bordPts : USINT; {DE:"Border thickness"}
	bordCol : UDINT; {DE:"Border color"}
	selBackCol : UDINT; {DE:"Selction background"}
	selForeCol : UDINT; {DE:"Selection foreground"}
	pRefrVar: UDINT; {DE:"Address of the refresh variable"}
	pSelVar : UDINT; {DE:"Address of the selection variable"}
	numChars : UINT; {DE:"Number of printable chars"}
	END_VAR

	VAR
	memVis : BOOL; {DE:"Visibility status"}
	END_VAR

	{CODE:EMBEDDED}

END_FUNCTION_BLOCK

FUNCTION_BLOCK Static02

	VAR_INPUT
	wHnd : UINT; {DE:"Object handle"}
	x : UINT; {DE:"X-coordinate of the upper-left corner"}
	y : UINT; {DE:"Y-coordinate of the upper-left corner"}
	accMode : USINT; {DE:"Access mode"}
	fResStr : BOOL; {DE:"Flag for resource strings"}
	pString : UDINT; {DE:"Address of the string"}
	pFont : UDINT; {DE:"Address of the font"}
	foreCol : UDINT; {DE:"Foreground color"}
	bckCol : UDINT; {DE:"Background color"}
	pVisVar : UDINT; {DE:"Address of the visibility flag"}
	format : UINT; {DE:"Alignment of static"}
	style : USINT; {DE:"Appearence"}
	bordPts : USINT; {DE:"Border thickness"}
	bordCol : UDINT; {DE:"Border color"}
	selBackCol : UDINT; {DE:"Selction background"}
	selForeCol : UDINT; {DE:"Selection foreground"}
	pRefrVar: UDINT; {DE:"Address of the refresh variable"}
	pSelVar : UDINT; {DE:"Address of the selection variable"}
	numChars : UINT; {DE:"Number of printable chars"}
	END_VAR

	VAR
	memVis : BOOL; {DE:"Visibility status"}
	pActString: UDINT; {DE:" Address of the string of the resource"}
	END_VAR

	{CODE:EMBEDDED}

END_FUNCTION_BLOCK

FUNCTION_BLOCK Image

	VAR_INPUT
	wHnd : UINT; {DE:"Object handle"}
	x1 : UINT; {DE:"X-coordinate of the upper-left corner"}
	y1 : UINT; {DE:"Y-coordinate of the upper-left corner"}
	px1 	 : UDINT; {DE:"Address of the variable X-coordinate of the upper-left corner"}
	py1 	 : UDINT; {DE:"Address of the variable Y-coordinate of the upper-left corner"}
	type_x 	 : USINT; {DE:"Data type of the X-coordinate variable"}
	type_y 	 : USINT; {DE:"Data type of the Y-coordinate variable"}
	dx : UINT; {DE:"X-coordinate of the lower-right corner"}
	dy : UINT; {DE:"Y-coordinate of the lower-right corner"}
	style : USINT; {DE:"Appearence"}
	floating : BOOL; {DE:"Floating style enabled"}
	bordPts : USINT; {DE:"Border thickness"}
	bordCol : UDINT; {DE:"Border color"}
	bordSelCol : UDINT; {DE:"Border selection color"}
	accMode : USINT; {DE:"Access mode"}
	pBmp : UDINT; {DE:"Address of the main bitmap"}
	pSelBmp : UDINT; {DE:"Address of the selection bitmap"}
	pSelVar : UDINT; {DE:"Address of the selection variable"}
	pVisVar : UDINT; {DE:"Address of the visibility variable"}
	END_VAR

	VAR_OUTPUT
	reqRefr : BOOL; {DE:"Request of refresh"}
	abs_x1 : UINT; {DE:"Absolute X-coordinate"}
	abs_y1 : UINT; {DE:"Absolute Y-coordinate"}
	mem_x1 : UINT; {DE:"Past absolute X-coordinate"}
	mem_y1 : UINT; {DE:"Past absolute Y-coordinate"}
	END_VAR

	VAR
	memVis : BOOL; {DE:"Visibility status"}
	memSel : BOOL; {DE:"Visibility status"}
	END_VAR

	{CODE:EMBEDDED}

END_FUNCTION_BLOCK

FUNCTION_BLOCK Image02

	VAR_INPUT
	wHnd : UINT; {DE:"Object handle"}
	x1 : UINT; {DE:"X-coordinate of the upper-left corner"}
	y1 : UINT; {DE:"Y-coordinate of the upper-left corner"}
	px1 	 : UDINT; {DE:"Address of the variable X-coordinate of the upper-left corner"}
	py1 	 : UDINT; {DE:"Address of the variable Y-coordinate of the upper-left corner"}
	type_x 	 : USINT; {DE:"Data type of the X-coordinate variable"}
	type_y 	 : USINT; {DE:"Data type of the Y-coordinate variable"}
	dx : UINT; {DE:"X-coordinate of the lower-right corner"}
	dy : UINT; {DE:"Y-coordinate of the lower-right corner"}
	style : USINT; {DE:"Appearence"}
	floating : BOOL; {DE:"Floating style enabled"}
	bordPts : USINT; {DE:"Border thickness"}
	bordCol : UDINT; {DE:"Border color"}
	bordSelCol : UDINT; {DE:"Border selection color"}
	accMode : USINT; {DE:"Access mode"}
	pBmp : UDINT; {DE:"Address of the main bitmap"}
	pVisVar : UDINT; {DE:"Address of the visibility variable"}
	END_VAR

	VAR_OUTPUT
	reqRefr : BOOL; {DE:"Request of refresh"}
	abs_x1 : UINT; {DE:"Absolute X-coordinate"}
	abs_y1 : UINT; {DE:"Absolute Y-coordinate"}
	mem_x1 : UINT; {DE:"Past absolute X-coordinate"}
	mem_y1 : UINT; {DE:"Past absolute Y-coordinate"}
	END_VAR

	VAR
	memVis : BOOL; {DE:"Visibility status"}
	pActualBmp : UDINT; {DE:"Visibility status"}
	END_VAR

	{CODE:EMBEDDED}

END_FUNCTION_BLOCK

FUNCTION_BLOCK Animation

	VAR_INPUT
	wHnd : UINT; {DE:"Object handle"}
	x1 : UINT; {DE:"X-coordinate of the upper-left corner"}
	y1 : UINT; {DE:"Y-coordinate of the upper-left corner"}
	x2 : UINT; {DE:"X-coordinate of the lower-right corner"}
	y2 : UINT; {DE:"Y-coordinate of the lower-right corner"}
	style : USINT; {DE:"Appearence"}
	bordPts  : USINT; {DE:"Border thickness"}
	bordCol  : UDINT; {DE:"Border color"}
	accMode  : USINT; {DE:"Access mode"}
	pBmpArr  : UDINT; {DE:"Address of the first element of the bitmap array"}
	pCaseArr : UDINT; {DE:"Address of the first element of the selection array"}
	nArrEl   : USINT; {DE:"Number of elements of the image list"}
	pBmpDef  : UDINT; {DE:"Address of the default bitmap"}
	pSelVar  : UDINT; {DE:"Address of the selection variable"}
	type 	 : USINT; {DE:"Data type of the selection variable"}
	pVisVar  : UDINT; {DE:"Address of the visibility variable"}
	END_VAR

	VAR
	mempBmp : UDINT; {DE:"Pointer to the bitmap drawn at the prev. iteration"}
	END_VAR

	{CODE:EMBEDDED}

END_FUNCTION_BLOCK

FUNCTION_BLOCK Animation02

	VAR_INPUT
	wHnd : UINT; {DE:"Object handle"}
	x1 : UINT; {DE:"X-coordinate of the upper-left corner"}
	y1 : UINT; {DE:"Y-coordinate of the upper-left corner"}
	x2 : UINT; {DE:"X-coordinate of the lower-right corner"}
	y2 : UINT; {DE:"Y-coordinate of the lower-right corner"}
	style : USINT; {DE:"Appearence"}
	bordPts  : USINT; {DE:"Border thickness"}
	bordCol  : UDINT; {DE:"Border color"}
	accMode  : USINT; {DE:"Access mode"}
	pBmpArr  : UDINT; {DE:"Address of the first element of the bitmap array"}
	pCaseArr : UDINT; {DE:"Address of the first element of the selection array"}
	nArrEl   : USINT; {DE:"Number of elements of the image list"}
	pBmpDef  : UDINT; {DE:"Address of the default bitmap"}
	pSelVar  : UDINT; {DE:"Address of the selection variable"}
	type 	 : USINT; {DE:"Data type of the selection variable"}
	pVisVar  : UDINT; {DE:"Address of the visibility variable"}
	END_VAR

	VAR
	mempBmp : UDINT; {DE:"Pointer to the bitmap drawn at the prev. iteration"}
	pActualBmpArr : UDINT;	{DE:"Address of the first element of the bitmap array "}
	pActualBmp: UDINT;	{DE:"Address of the actual bitmap"}
	pActualBmpDef: UDINT;	{DE:"Address of the actual default bitmap"}
	END_VAR

	{CODE:EMBEDDED}

END_FUNCTION_BLOCK

FUNCTION_BLOCK Button01

	VAR_INPUT
	wHnd : UINT; {DE:"Object handle"}
	x1 : UINT; {DE:"X-coordinate of the upper-left corner"}
	y1 : UINT; {DE:"Y-coordinate of the upper-left corner"}
	x2 : UINT; {DE:"X-coordinate of the lower-right corner"}
	y2 : UINT; {DE:"Y-coordinate of the lower-right corner"}
	fResStr : BOOL; {DE:"Flag for resource strings"}
	pText : UDINT; {DE:"Address of the foreground string / picture"}
	pFont : UDINT; {DE:"Address of the font"}
	style : USINT; {DE:"Appearence"}
	bordPts : USINT; {DE:"Border thickness"}
	bordCol : UDINT; {DE:"Border color"}
	fillCol : UDINT; {DE:"Fill color"}
	bordSelCol : UDINT; {DE:"Border selection color"}
	fillSelCol : UDINT; {DE:"Fill selection color"}
	accMode : USINT; {DE:"Access mode"}
	pVisVar : UDINT; {DE:"Address of the visibility variable"}
	pTransp : UDINT; {DE:"Address of the transparency variable"}
	pPressVar : UDINT; {DE:"Address of the pressure variable"}
	pSelVar : UDINT; {DE:"Address of the selection variable"}
	pSelText : UDINT; {DE:"Address of the selection string / picture"}
	format : UINT; {DE:"Control word"}
	END_VAR

	VAR
	memVis : BOOL; {DE:"Visibility status"}
	memTransp : BOOL; {DE:"Transparency status"}
	memSel : BOOL; {DE:"Transparency status"}
	END_VAR

	{CODE:EMBEDDED}

END_FUNCTION_BLOCK

FUNCTION_BLOCK Button02

	VAR_INPUT
	wHnd : UINT; {DE:"Object handle"}
	x1 : UINT; {DE:"X-coordinate of the upper-left corner"}
	y1 : UINT; {DE:"Y-coordinate of the upper-left corner"}
	x2 : UINT; {DE:"X-coordinate of the lower-right corner"}
	y2 : UINT; {DE:"Y-coordinate of the lower-right corner"}
	fResStr : BOOL; {DE:"Flag for resource strings"}
	pText : UDINT; {DE:"Address of the foreground string / picture"}
	pFont : UDINT; {DE:"Address of the font"}
	style : USINT; {DE:"Appearence"}
	bordPts : USINT; {DE:"Border thickness"}
	bordCol : UDINT; {DE:"Border color"}
	fillCol : UDINT; {DE:"Fill color"}
	bordSelCol : UDINT; {DE:"Border selection color"}
	fillSelCol : UDINT; {DE:"Fill selection color"}
	accMode : USINT; {DE:"Access mode"}
	pVisVar : UDINT; {DE:"Address of the visibility variable"}
	pTransp : UDINT; {DE:"Address of the transparency variable"}
	pPressVar : UDINT; {DE:"Address of the pressure variable"}
	pSelVar : UDINT; {DE:"Address of the selection variable"}
	pSelText : UDINT; {DE:"Address of the selection string / picture"}
	format : UINT; {DE:"Control word"}
	order : UINT; {DE:"Selection Order"}
	END_VAR

	VAR
	memVis : BOOL; {DE:"Visibility status"}
	memTransp : BOOL; {DE:"Transparency status"}
	memSel : BOOL; {DE:"Transparency status"}
	END_VAR

	{CODE:EMBEDDED}

END_FUNCTION_BLOCK

FUNCTION_BLOCK Button03

	VAR_INPUT
	wHnd : UINT; {DE:"Object handle"}
	x1 : UINT; {DE:"X-coordinate of the upper-left corner"}
	y1 : UINT; {DE:"Y-coordinate of the upper-left corner"}
	x2 : UINT; {DE:"X-coordinate of the lower-right corner"}
	y2 : UINT; {DE:"Y-coordinate of the lower-right corner"}
	fResStr : BOOL; {DE:"Flag for resource strings"}
	pText : UDINT; {DE:"Address of the foreground string / picture"}
	pFont : UDINT; {DE:"Address of the font"}
	style : USINT; {DE:"Appearence"}
	bordPts : USINT; {DE:"Border thickness"}
	bordCol : UDINT; {DE:"Border color"}
	fillCol : UDINT; {DE:"Fill color"}
	bordSelCol : UDINT; {DE:"Border selection color"}
	fillSelCol : UDINT; {DE:"Fill selection color"}
	accMode : USINT; {DE:"Access mode"}
	pVisVar : UDINT; {DE:"Address of the visibility variable"}
	pTransp : UDINT; {DE:"Address of the transparency variable"}
	pPressVar : UDINT; {DE:"Address of the pressure variable"}
	pSelVar : UDINT; {DE:"Address of the selection variable"}
	pSelText : UDINT; {DE:"Address of the selection string / picture"}
	format : UINT; {DE:"Control word"}
	order : UINT; {DE:"Selection Order"}
	type : USINT; {DE:"Type (normal, toggle)"}
	END_VAR

	VAR
	memVis : BOOL; {DE:"Visibility status"}
	memTransp : BOOL; {DE:"Transparency status"}
	memSel : BOOL; {DE:"Transparency status"}
	END_VAR

	{CODE:EMBEDDED}

END_FUNCTION_BLOCK

FUNCTION_BLOCK Button04

VAR_INPUT
	wHnd : UINT;		{DE:"Object handle"}
	x1 : UINT;			{DE:"X-coordinate of the upper-left corner"}
	y1 : UINT;			{DE:"Y-coordinate of the upper-left corner"}
	x2 : UINT;			{DE:"X-coordinate of the lower-right corner"}
	y2 : UINT;			{DE:"Y-coordinate of the lower-right corner"}
	pText : UDINT;		{DE:"Address of the foreground string"}
	pImage : UDINT;		{DE:"Address of the foreground picture"}
	pFont : UDINT;		{DE:"Address of the font"}
	style : USINT;		{DE:"Appearence"}
	bordPts : USINT;	{DE:"Border thickness"}
	textCol : UDINT;	{DE:"Text color"}
	bordCol : UDINT;	{DE:"Border color"}
	fillCol : UDINT;	{DE:"Fill color"}
	textSelCol : UDINT;	{DE:"Text selection color"}
	bordSelCol : UDINT;	{DE:"Border selection color"}
	fillSelCol : UDINT;	{DE:"Fill selection color"}
	accMode : USINT;	{DE:"Access mode"}
	pVisVar : UDINT;	{DE:"Address of the visibility variable"}
	pPressVar : UDINT;	{DE:"Address of the pressure variable"}
	pSelVar : UDINT;	{DE:"Address of the selection variable"}
	pSelText : UDINT;	{DE:"Address of the selection string"}
	pSelImage : UDINT;	{DE:"Address of the selection picture"}
	format : UINT;		{DE:"Control word"}
	order : UINT;		{DE:"Selection Order"}
	type : USINT;		{DE:"Type (normal, toggle)"}
END_VAR

VAR
	memVis : BOOL;		{DE:"Visibility status"}
	memSel : BOOL;		{DE:"Transparency status"}
END_VAR

	{CODE:EMBEDDED}

END_FUNCTION_BLOCK

FUNCTION_BLOCK Button05

	VAR_INPUT
	wHnd : UINT; {DE:"Object handle"}
	x1 : UINT; {DE:"X-coordinate of the upper-left corner"}
	y1 : UINT; {DE:"Y-coordinate of the upper-left corner"}
	x2 : UINT; {DE:"X-coordinate of the lower-right corner"}
	y2 : UINT; {DE:"Y-coordinate of the lower-right corner"}
	pText : UDINT;		{DE:"Address of the foreground string"}
	pImage : UDINT;		{DE:"Address of the foreground picture"}
	pFont : UDINT; {DE:"Address of the font"}
	style : USINT; {DE:"Appearence"}
	bordPts : USINT; {DE:"Border thickness"}
	textCol : UDINT;	{DE:"Text color"}
	bordCol : UDINT; {DE:"Border color"}
	fillCol : UDINT; {DE:"Fill color"}
	textSelCol : UDINT;	{DE:"Text selection color"}
	bordSelCol : UDINT; {DE:"Border selection color"}
	fillSelCol : UDINT; {DE:"Fill selection color"}
	accMode : USINT; {DE:"Access mode"}
	pVisVar : UDINT; {DE:"Address of the visibility variable"}
	pPressVar : UDINT; {DE:"Address of the pressure variable"}
	pSelVar : UDINT; {DE:"Address of the selection variable"}
	pSelText : UDINT;	{DE:"Address of the selection string"}
	pSelImage : UDINT;	{DE:"Address of the selection picture"}
	format : UINT; {DE:"Control word"}
	order : UINT; {DE:"Selection Order"}
	type : USINT; {DE:"Type (normal, toggle)"}
	END_VAR

	VAR
	memVis : BOOL; {DE:"Visibility status"}
	memSel : BOOL; 	{DE:"Transparency status"}
	pActSelText: UDINT; {DE:" Address of the selection string now "}
	pActText: UDINT;	{DE:" Address of the foreground string now"}
	pActImage: UDINT;	{DE:" Address of the foreground picture "}
	pActSelImage: UDINT; {DE:" Address of the selection picture "}
	END_VAR

	{CODE:EMBEDDED}

END_FUNCTION_BLOCK

FUNCTION_BLOCK CheckBox01

	VAR_INPUT
		pVar : UDINT;		{ DE:"Address of the associated variable" }
		pVisVar : UDINT;	{ DE:"Address of the visibility variable" }
		pSelVar : UDINT;	{ DE:"Address of the selectability variable" }
		foreCol : UDINT;	{ DE:"Foreground color" }
		bckCol : UDINT;		{ DE:"Background color" }
		foreSelCol : UDINT;	{ DE:"Foreground selection color" }
		bckSelCol : UDINT;	{ DE:"Background selection color" }
		bordCol : UDINT;	{ DE:"Border color" }
		wHnd : UINT;		{ DE:"Object handle" }
		x1 : UINT;		{ DE:"X-coordinate of the upper-left corner" }
		y1 : UINT;		{ DE:"Y-coordinate of the upper-left corner" }
		x2 : UINT;		{ DE:"X-coordinate of the lower-right corner" }
		y2 : UINT;		{ DE:"Y-coordinate of the lower-right corner" }
		style : USINT;		{ DE:"Appearence" }
		tickStyle : USINT;	{ DE:"Tick style" }
		bordPts : USINT;	{ DE:"Border thickness" }
		order : USINT;		{ DE:"Selection order" }
		accMode : USINT;	{ DE:"Access mode" }
		rw : USINT;		{ DE:"Flag of write-mode enabled" }
		isParam : USINT;	{ DE:"Parameter/Normal variable" }
	END_VAR

	VAR
		memValue : USINT;	{ DE:"Preceding value" }
		memVis : USINT;		{ DE:"Visibility status" }
		memSel : USINT;		{ DE:"Selection status" }
		spare8 : USINT;		{ DE:"Spare data" }
	END_VAR

	{CODE:EMBEDDED}

END_FUNCTION_BLOCK

FUNCTION_BLOCK CheckBox02

	VAR_INPUT
		pVar : UDINT;		{ DE:"Address of the associated variable" }
		pVisVar : UDINT;	{ DE:"Address of the visibility variable" }
		pSelVar : UDINT;	{ DE:"Address of the selectability variable" }
		foreCol : UDINT;	{ DE:"Foreground color" }
		bckCol : UDINT;		{ DE:"Background color" }
		foreSelCol : UDINT;	{ DE:"Foreground selection color" }
		bckSelCol : UDINT;	{ DE:"Background selection color" }
		bordCol : UDINT;	{ DE:"Border color" }
		wHnd : UINT;		{ DE:"Object handle" }
		x1 : UINT;		{ DE:"X-coordinate of the upper-left corner" }
		y1 : UINT;		{ DE:"Y-coordinate of the upper-left corner" }
		x2 : UINT;		{ DE:"X-coordinate of the lower-right corner" }
		y2 : UINT;		{ DE:"Y-coordinate of the lower-right corner" }
		style : USINT;		{ DE:"Appearence" }
		tickStyle : USINT;	{ DE:"Tick style" }
		bordPts : USINT;	{ DE:"Border thickness" }
		order : USINT;		{ DE:"Selection order" }
		accMode : USINT;	{ DE:"Access mode" }
		rw : USINT;		{ DE:"Flag of write-mode enabled" }
		isParam : USINT;	{ DE:"Parameter/Normal variable" }
	END_VAR

	VAR
		memValue : USINT;	{ DE:"Preceding value" }
		memVis : USINT;		{ DE:"Visibility status" }
		memSel : USINT;		{ DE:"Selection status" }
		spare8 : USINT;		{ DE:"Spare data" }
		pValue : UDINT;		{ DE: "Pointer to the value - only for HMIRuntimeCore" }
		pInfoRec : UDINT;	{ DE: "Pointer to the record with remote param info - only for HMIRuntimeCore" }
	END_VAR

	{CODE:EMBEDDED}

END_FUNCTION_BLOCK

FUNCTION_BLOCK EditBox01

	VAR_INPUT
	wHnd : UINT; {DE:"Object handle"}
	x1 : UINT; {DE:"X-coordinate of the upper-left corner"}
	y1 : UINT; {DE:"Y-coordinate of the upper-left corner"}
	x2 : UINT; {DE:"X-coordinate of the lower-right corner"}
	y2 : UINT; {DE:"Y-coordinate of the lower-right corner"}
	pFont : UDINT; {DE:"Address of the font"}
	style : USINT; {DE:"Appearence"}
	foreCol : UDINT; {DE:"Foreground color"}
	bckCol : UDINT; {DE:"Background color"}
	foreSelCol : UDINT; {DE:"Foreground selection color"}
	bckSelCol : UDINT; {DE:"Background selection color"}
	bordPts : USINT; {DE:"Border thickness"}
	bordCol : UDINT; {DE:"Border color"}
	rw : BOOL; {DE:"Flag of write-mode enabled"}
	refr : BOOL; {DE:"Flag of refresh required"}
	pVar : UDINT; {DE:"Address of the associated variable"}
	type : USINT; {DE:"Data type of the associated variable"}
	pVarMin : UDINT; {DE:"Address of the lower limit variable"}
	pVarMax : UDINT; {DE:"Address of the higher limit variable"}
	enumId : INT; {DE:"Identifier of the associated enumerated data type"}
	format : UDINT; {DE:"Format code"}
	pVisVar : UDINT; {DE:"Address of the visibility variable"}
	pCanSel : UDINT; {DE:"Address of the selectability variable"}
	order : USINT; {DE:"Selection order"}
	accMode : USINT; {DE:"Access mode"}
	END_VAR

	VAR_OUTPUT
	outKey : SINT; {DE:"Key pressed to exit the edit mode"}
	END_VAR

	VAR
	memVis : BOOL; {DE:"Visibility status"}
	END_VAR

	{CODE:EMBEDDED}

END_FUNCTION_BLOCK

FUNCTION_BLOCK EditBox02

	VAR_INPUT
	wHnd : UINT; {DE:"Object handle"}
	x1 : UINT; {DE:"X-coordinate of the upper-left corner"}
	y1 : UINT; {DE:"Y-coordinate of the upper-left corner"}
	x2 : UINT; {DE:"X-coordinate of the lower-right corner"}
	y2 : UINT; {DE:"Y-coordinate of the lower-right corner"}
	pFont : UDINT; {DE:"Address of the font"}
	style : USINT; {DE:"Appearence"}
	foreCol : UDINT; {DE:"Foreground color"}
	bckCol : UDINT; {DE:"Background color"}
	foreSelCol : UDINT; {DE:"Foreground selection color"}
	bckSelCol : UDINT; {DE:"Background selection color"}
	bordPts : USINT; {DE:"Border thickness"}
	bordCol : UDINT; {DE:"Border color"}
	rw : BOOL; {DE:"Flag of write-mode enabled"}
	refr : BOOL; {DE:"Flag of refresh required"}
	pVar : UDINT; {DE:"Address of the associated variable"}
	type : USINT; {DE:"Data type of the associated variable"}
	pVarMin : UDINT; {DE:"Address of the lower limit variable"}
	pVarMax : UDINT; {DE:"Address of the higher limit variable"}
	enumId : INT; {DE:"Identifier of the associated enumerated data type"}
	format : UDINT; {DE:"Format code"}
	pVisVar : UDINT; {DE:"Address of the visibility variable"}
	pCanSel : UDINT; {DE:"Address of the selectability variable"}
	order : USINT; {DE:"Selection order"}
	accMode : USINT; {DE:"Access mode"}
	pLabel : UDINT; {DE:"Description"}
	END_VAR

	VAR_OUTPUT
	outKey : SINT; {DE:"Key pressed to exit the edit mode"}
	END_VAR

	VAR
	memVis : BOOL; {DE:"Visibility status"}
	pValue : UDINT; {DE: "Pointer to the value - only for HMIRuntimeCore" }
	pInfoRec : UDINT; {DE: "Pointer to the record with remote param info - only for HMIRuntimeCore" }
	END_VAR

	{CODE:EMBEDDED}

END_FUNCTION_BLOCK

FUNCTION_BLOCK EditBox03

	VAR_INPUT
	wHnd : UINT; {DE:"Object handle"}
	x1 : UINT; {DE:"X-coordinate of the upper-left corner"}
	y1 : UINT; {DE:"Y-coordinate of the upper-left corner"}
	x2 : UINT; {DE:"X-coordinate of the lower-right corner"}
	y2 : UINT; {DE:"Y-coordinate of the lower-right corner"}
	pFont : UDINT; {DE:"Address of the font"}
	style : USINT; {DE:"Appearence"}
	foreCol : UDINT; {DE:"Foreground color"}
	bckCol : UDINT; {DE:"Background color"}
	foreSelCol : UDINT; {DE:"Foreground selection color"}
	bckSelCol : UDINT; {DE:"Background selection color"}
	bordPts : USINT; {DE:"Border thickness"}
	bordCol : UDINT; {DE:"Border color"}
	rw : BOOL; {DE:"Flag of write-mode enabled"}
	refr : BOOL; {DE:"Flag of refresh required"}
	pVar : UDINT; {DE:"Address of the associated variable"}
	type : USINT; {DE:"Data type of the associated variable"}
	pVarMin : UDINT; {DE:"Address of the lower limit variable"}
	pVarMax : UDINT; {DE:"Address of the higher limit variable"}
	format : UDINT; {DE:"Format code"}
	pVisVar : UDINT; {DE:"Address of the visibility variable"}
	pCanSel : UDINT; {DE:"Address of the selectability variable"}
	order : USINT; {DE:"Selection order"}
	accMode : USINT; {DE:"Access mode"}
	pLabel : UDINT; {DE:"Description"}
	pEnumId: UDINT; {DE:"Enum id"}
	END_VAR

	VAR_OUTPUT
	outKey : SINT; {DE:"Key pressed to exit the edit mode"}
	END_VAR

	VAR
	memVis : BOOL; {DE:"Visibility status"}
	pValue : UDINT; {DE: "Pointer to the value - only for HMIRuntimeCore" }
	pInfoRec : UDINT; {DE: "Pointer to the record with remote param info - only for HMIRuntimeCore" }
	pEnumRec : UDINT; {DE: "Pointer to the record of enum selected" }
	END_VAR

	{CODE:EMBEDDED}

END_FUNCTION_BLOCK

FUNCTION_BLOCK ComboBox01

	VAR_INPUT
		pVar : UDINT;		{ DE:"Address of the associated variable" }
		pVisVar : UDINT;	{ DE:"Address of the visibility variable" }
		pSelVar : UDINT;	{ DE:"Address of the selectability variable" }
		pFont : UDINT;		{ DE:"Address of the font" }
		foreCol : UDINT;	{ DE:"Foreground color" }
		bckCol : UDINT;		{ DE:"Background color" }
		foreSelCol : UDINT;	{ DE:"Foreground selection color" }
		bckSelCol : UDINT;	{ DE:"Background selection color" }
		bordCol : UDINT;	{ DE:"Border color" }
		wHnd : UINT;		{ DE:"Object handle" }
		x1 : UINT;		{ DE:"X-coordinate of the upper-left corner" }
		y1 : UINT;		{ DE:"Y-coordinate of the upper-left corner" }
		x2 : UINT;		{ DE:"X-coordinate of the lower-right corner" }
		y2 : UINT;		{ DE:"Y-coordinate of the lower-right corner" }
		enumId : INT;		{ DE:"Identifier of the associated enumerated data type" }
		style : USINT;		{ DE:"Appearence" }
		bordPts : USINT;	{ DE:"Border thickness" }
		order : USINT;		{ DE:"Selection order" }
		accMode : USINT;	{ DE:"Access mode" }
		rw : USINT;		{ DE:"Flag of write-mode enabled" }
		isParam : USINT;	{ DE:"Parameter/Normal variable" }
		type : USINT;	{ DE:"Data type of the associated variable" }
	END_VAR

	VAR_OUTPUT
		outKey : SINT;		{ DE:"Key pressed to exit the edit mode" }
	END_VAR

	VAR
		memValue : DINT;	{ DE:"Preceding value" }
		memVis : USINT;		{ DE:"Visibility status" }
		memSel : USINT;		{ DE:"Selection status" }
		spare16 : UINT;		{ DE:"Spare data" }
	END_VAR

	{CODE:EMBEDDED}

END_FUNCTION_BLOCK

FUNCTION_BLOCK ComboBox02

	VAR_INPUT
		pVar : UDINT;		{ DE:"Address of the associated variable" }
		pVisVar : UDINT;	{ DE:"Address of the visibility variable" }
		pSelVar : UDINT;	{ DE:"Address of the selectability variable" }
		pFont : UDINT;		{ DE:"Address of the font" }
		foreCol : UDINT;	{ DE:"Foreground color" }
		bckCol : UDINT;		{ DE:"Background color" }
		foreSelCol : UDINT;	{ DE:"Foreground selection color" }
		bckSelCol : UDINT;	{ DE:"Background selection color" }
		bordCol : UDINT;	{ DE:"Border color" }
		wHnd : UINT;		{ DE:"Object handle" }
		x1 : UINT;		{ DE:"X-coordinate of the upper-left corner" }
		y1 : UINT;		{ DE:"Y-coordinate of the upper-left corner" }
		x2 : UINT;		{ DE:"X-coordinate of the lower-right corner" }
		y2 : UINT;		{ DE:"Y-coordinate of the lower-right corner" }
		enumId : INT;		{ DE:"Identifier of the associated enumerated data type" }
		style : USINT;		{ DE:"Appearence" }
		bordPts : USINT;	{ DE:"Border thickness" }
		order : USINT;		{ DE:"Selection order" }
		accMode : USINT;	{ DE:"Access mode" }
		rw : USINT;		{ DE:"Flag of write-mode enabled" }
		isParam : USINT;	{ DE:"Parameter/Normal variable" }
		type : USINT;	{ DE:"Data type of the associated variable" }
	END_VAR

	VAR_OUTPUT
		outKey : SINT;		{ DE:"Key pressed to exit the edit mode" }
	END_VAR

	VAR
		memValue : DINT;	{ DE:"Preceding value" }
		memVis : USINT;		{ DE:"Visibility status" }
		memSel : USINT;		{ DE:"Selection status" }
		spare16 : UINT;		{ DE:"Spare data" }
		pValue : UDINT;		{ DE: "Pointer to the value - only for HMIRuntimeCore" }
		pInfoRec : UDINT;	{ DE: "Pointer to the record with remote param info - only for HMIRuntimeCore" }
	END_VAR

	{CODE:EMBEDDED}

END_FUNCTION_BLOCK

FUNCTION_BLOCK ComboBox03

	VAR_INPUT
		pVar : UDINT;		{ DE:"Address of the associated variable" }
		pVisVar : UDINT;	{ DE:"Address of the visibility variable" }
		pSelVar : UDINT;	{ DE:"Address of the selectability variable" }
		pFont : UDINT;		{ DE:"Address of the font" }
		foreCol : UDINT;	{ DE:"Foreground color" }
		bckCol : UDINT;		{ DE:"Background color" }
		foreSelCol : UDINT;	{ DE:"Foreground selection color" }
		bckSelCol : UDINT;	{ DE:"Background selection color" }
		bordCol : UDINT;	{ DE:"Border color" }
		wHnd : UINT;		{ DE:"Object handle" }
		x1 : UINT;		{ DE:"X-coordinate of the upper-left corner" }
		y1 : UINT;		{ DE:"Y-coordinate of the upper-left corner" }
		x2 : UINT;		{ DE:"X-coordinate of the lower-right corner" }
		y2 : UINT;		{ DE:"Y-coordinate of the lower-right corner" }
		style : USINT;		{ DE:"Appearence" }
		bordPts : USINT;	{ DE:"Border thickness" }
		order : USINT;		{ DE:"Selection order" }
		accMode : USINT;	{ DE:"Access mode" }
		rw : USINT;		{ DE:"Flag of write-mode enabled" }
		isParam : USINT;	{ DE:"Parameter/Normal variable" }
		type : USINT;	{ DE:"Data type of the associated variable" }
		pEnumId: UDINT;	{ DE:" Pointer to the strings of the id enum" }
	END_VAR

	VAR_OUTPUT
		outKey : SINT;		{ DE:"Key pressed to exit the edit mode" }
	END_VAR

	VAR
		memValue : DINT;	{ DE:"Preceding value" }
		memVis : USINT;		{ DE:"Visibility status" }
		memSel : USINT;		{ DE:"Selection status" }
		spare16 : UINT;		{ DE:"Spare data" }
		pValue : UDINT;		{ DE: "Pointer to the value - only for HMIRuntimeCore" }
		pInfoRec : UDINT;	{ DE: "Pointer to the record with remote param info - only for HMIRuntimeCore" }
		pEnumRec: UDINT;	{ DE:"Pointer to the record of the selected enum" }
	END_VAR

	{CODE:EMBEDDED}

END_FUNCTION_BLOCK

FUNCTION_BLOCK Progress

	VAR_INPUT
	wHnd : UINT; {DE:"Object handle"}
	x1 : UINT; {DE:"X-coordinate of the upper-left corner"}
	y1 : UINT; {DE:"Y-coordinate of the upper-left corner"}
	x2 : UINT; {DE:"X-coordinate of the lower-right corner"}
	y2 : UINT; {DE:"Y-coordinate of the lower-right corner"}
	style : USINT; {DE:"Appearence"}
	barCol : UDINT; {DE:"Bar color"}
	bckCol : UDINT; {DE:"Background color"}
	bordPts : USINT; {DE:"Border thickness"}
	bordCol : UDINT; {DE:"Border color"}
	pVar : UDINT; {DE:"Address of the associated variable"}
	type : USINT; {DE:"Data type of the associated variable"}
	pMin : UDINT; {DE:"Address of the lower bound"}
	pMax : UDINT; {DE:"Address of the higher bound"}
	format : UDINT; {DE:"Format code"}
	pVisVar : UDINT; {DE:"Address of the visibility variable"}
	accMode : USINT; {DE:"Access mode"}
	END_VAR

	VAR
	memVal : UDINT; {DE:"Progress status"}
	memVis : BOOL; {DE:"Visibility status"}
	END_VAR

	{CODE:EMBEDDED}

END_FUNCTION_BLOCK

FUNCTION_BLOCK Progress02

	VAR_INPUT
	wHnd : UINT; {DE:"Object handle"}
	x1 : UINT; {DE:"X-coordinate of the upper-left corner"}
	y1 : UINT; {DE:"Y-coordinate of the upper-left corner"}
	x2 : UINT; {DE:"X-coordinate of the lower-right corner"}
	y2 : UINT; {DE:"Y-coordinate of the lower-right corner"}
	style : USINT; {DE:"Appearence"}
	barCol : UDINT; {DE:"Bar color"}
	bckCol : UDINT; {DE:"Background color"}
	bordPts : USINT; {DE:"Border thickness"}
	bordCol : UDINT; {DE:"Border color"}
	pVar : UDINT; {DE:"Address of the associated variable"}
	type : USINT; {DE:"Data type of the associated variable"}
	pMin : UDINT; {DE:"Address of the lower bound"}
	pMax : UDINT; {DE:"Address of the higher bound"}
	format : UDINT; {DE:"Format code"}
	pVisVar : UDINT; {DE:"Address of the visibility variable"}
	accMode : USINT; {DE:"Access mode"}
	END_VAR

	VAR
	memVal : UDINT; {DE:"Progress status"}
	memVis : BOOL; {DE:"Visibility status"}
	pValue : UDINT; {DE: "Pointer to the value - only for HMIRuntimeCore" }
	pInfoRec : UDINT; {DE: "Pointer to the record with remote param info - only for HMIRuntimeCore" }
	END_VAR

	{CODE:EMBEDDED}

END_FUNCTION_BLOCK

FUNCTION_BLOCK Chart

	VAR_INPUT
	wHnd : UINT; {DE:"Object handle"}
	x1 : UINT; {DE:"X-coordinate of the upper-left corner"}
	y1 : UINT; {DE:"Y-coordinate of the upper-left corner"}
	x2 : UINT; {DE:"X-coordinate of the lower-right corner"}
	y2 : UINT; {DE:"Y-coordinate of the lower-right corner"}
	pFont : UDINT; {DE:"Address of the font"}
	style : USINT; {DE:"Appearence"}
	bordPts : USINT; {DE:"Border thickness"}
	bordCol : UDINT; {DE:"Border color"}
	backCol : UDINT; {DE:"Background color"}
	tyNSamples : UINT; {DE:"Type of Number of samples"}
	pNSamples :  UDINT; {DE:"Number of samples"}
	tyXOffset : UINT;  {DE:"Type of X Offset"}
	pXOffset: UDINT; {DE:"X Offset"}
	tyTrackRight : UINT; {DE:"Right label track type"}
	pTrackRight : UDINT; {DE:"Right label track"}
	tyTrackLeft : UINT; {DE:"Left label track type"}
	pTrackLeft : UDINT; {DE:"left label track"}
	formatLeft :  UDINT; {DE:"format of Y label left"}
	formatRight :  UDINT; {DE:"format of Y label right "}
	fGrid : BOOL; {DE:"Flag for grid display"}
	iDivGridX : UINT; {DE:"Horizontal divisions"}
	iDivGridY : UINT; {DE:"Vertical divisions"}
	accMode : USINT; {DE:"Access mode"}
	iXLabelDiv : UINT; {DE:"How many x label"}
	tyXScaleType : UINT; {DE:"X Scale type"}
	pXScale : UDINT; {DE:"X Scale"}
	pClearVar : UDINT; {DE:"Variabile di clear dei dati"}
	pVisVar : UDINT; {DE:"Address of the visibility variable"}
	pRefrVar: UDINT; {DE:"Address of the refresh variable"}
	format :  UDINT; {DE:"format of X labels"}
	pXData :  UDINT; {DE:"pointer to X data"}
	tyXData : UINT; {DE:"type of X data"}
	XLabelCol : UDINT;{DE:"Color of X label"}
	iDotStep: UINT; {DE:"distance between points of grid"}
	iSampleBuffer: UINT; {DE:" size of sample buffer "}
	arXBars :  ARRAY [0..2] OF UDINT; {DE:"X Bars"}
	arXBarsType : ARRAY [0..2] OF UINT; {DE:"Type of data of X Bars"}
	arXBarsCol: ARRAY [0..2] OF UDINT; {DE:"Bars colors"}
	GridCol : UDINT;	{DE:"Grid color "}
	BorderGridCol : UDINT;	{DE:"Border grid color "}
	arTrkData : ARRAY [0..7] OF UDINT; {DE:"Array of track data addresses"}
	arTrkType : ARRAY [0..7] OF USINT; {DE:"Data type of the associated variable"}
	arTrkCol : ARRAY [0..7] OF UDINT; {DE:"Array of track colors"}
	arTrkScaleY : ARRAY [0..7] OF UDINT;   {DE:"Array of track scale"}
	arTrkScaleYType: ARRAY [0..7] OF UINT; {DE:"Array of track scale type"}
	arTrkOffset: ARRAY [0..7] OF UDINT;    {DE:"Array of track offset"}
	arTrkOffsetType: ARRAY [0..7] OF UINT; {DE:"Array of track offset type"}
	arTrkVis : ARRAY [0..7] OF UDINT; {DE:"Array of track visibility variables"}
	iYLabelDiv: ARRAY [0..7] OF UINT; {DE:"Array of vertical label"}
	arTrkBarValue: ARRAY [0..23] OF UDINT; {DE:"Array of value of horizontal bar"}
	arTrkBarValueType: ARRAY [0..23] OF UINT; {DE:"Array of value of horizontal bar"}
	arTrkBarName: ARRAY [0..23] OF UDINT; {DE:"Array of names of horizontal bar"}
	arTrkBarCol: ARRAY [0..23] OF UDINT; {DE:"Array of colors of horizontal bar"}
	arTrkMinScale: ARRAY [0..23] OF UDINT; {DE:"Array of min scale y acceptable"}
	END_VAR

	VAR
	memVis : BOOL; {DE:"Visibility status"}
	grx1 : UINT; {DE:"X-coordinate of the upper-left corner of the active area"}
	gry1 : UINT; {DE:"Y-coordinate of the upper-left corner of the active area"}
	grx2 : UINT; {DE:"X-coordinate of the lower-right corner of the active area"}
	gry2 : UINT; {DE:"Y-coordinate of the lower-right corner of the active area"}
	pChart : DWORD; {DE:"Address of the chart"}
	lastIdxSamples: UDINT; {DE:" last index of the array of samples "}

	END_VAR

	{CODE:EMBEDDED}

END_FUNCTION_BLOCK

FUNCTION_BLOCK Chart02

	VAR_INPUT
	wHnd : UINT; {DE:"Object handle"}
	x1 : UINT; {DE:"X-coordinate of the upper-left corner"}
	y1 : UINT; {DE:"Y-coordinate of the upper-left corner"}
	x2 : UINT; {DE:"X-coordinate of the lower-right corner"}
	y2 : UINT; {DE:"Y-coordinate of the lower-right corner"}
	pFont : UDINT; {DE:"Address of the font"}
	style : USINT; {DE:"Appearence"}
	bordPts : USINT; {DE:"Border thickness"}
	bordCol : UDINT; {DE:"Border color"}
	backCol : UDINT; {DE:"Background color"}
	tyNSamples : UINT; {DE:"Type of Number of samples"}
	pNSamples :  UDINT; {DE:"Number of samples"}
	tyXOffset : UINT;  {DE:"Type of X Offset"}
	pXOffset: UDINT; {DE:"X Offset"}
	tyTrackRight : UINT; {DE:"Right label track type"}
	pTrackRight : UDINT; {DE:"Right label track"}
	tyTrackLeft : UINT; {DE:"Left label track type"}
	pTrackLeft : UDINT; {DE:"left label track"}
	formatLeft :  UDINT; {DE:"format of Y label left"}
	formatRight :  UDINT; {DE:"format of Y label right "}
	fGrid : BOOL; {DE:"Flag for grid display"}
	iDivGridX : UINT; {DE:"Horizontal divisions"}
	iDivGridY : UINT; {DE:"Vertical divisions"}
	accMode : USINT; {DE:"Access mode"}
	iXLabelDiv : UINT; {DE:"How many x label"}
	tyXScaleType : UINT; {DE:"X Scale type"}
	pXScale : UDINT; {DE:"X Scale"}
	pClearVar : UDINT; {DE:"Variabile di clear dei dati"}
	pVisVar : UDINT; {DE:"Address of the visibility variable"}
	pRefrVar: UDINT; {DE:"Address of the refresh variable"}
	format :  UDINT; {DE:"format of X labels"}
	pXData :  UDINT; {DE:"pointer to X data"}
	tyXData : UINT; {DE:"type of X data"}
	XLabelCol : UDINT;{DE:"Color of X label"}
	iDotStep: UINT; {DE:"distance between points of grid"}
	iSampleBuffer: UDINT; {DE:" size of sample buffer "}
	arXBars :  ARRAY [0..2] OF UDINT; {DE:"X Bars"}
	arXBarsType : ARRAY [0..2] OF UINT; {DE:"Type of data of X Bars"}
	arXBarsCol: ARRAY [0..2] OF UDINT; {DE:"Bars colors"}
	GridCol : UDINT;	{DE:"Grid color "}
	BorderGridCol : UDINT;	{DE:"Border grid color "}
	arTrkData : ARRAY [0..7] OF UDINT; {DE:"Array of track data addresses"}
	arTrkType : ARRAY [0..7] OF USINT; {DE:"Data type of the associated variable"}
	arTrkCol : ARRAY [0..7] OF UDINT; {DE:"Array of track colors"}
	arTrkScaleY : ARRAY [0..7] OF UDINT;   {DE:"Array of track scale"}
	arTrkScaleYType: ARRAY [0..7] OF UINT; {DE:"Array of track scale type"}
	arTrkOffset: ARRAY [0..7] OF UDINT;    {DE:"Array of track offset"}
	arTrkOffsetType: ARRAY [0..7] OF UINT; {DE:"Array of track offset type"}
	arTrkVis : ARRAY [0..7] OF UDINT; {DE:"Array of track visibility variables"}
	iYLabelDiv: ARRAY [0..7] OF UINT; {DE:"Array of vertical label"}
	arTrkBarValue: ARRAY [0..23] OF UDINT; {DE:"Array of value of horizontal bar"}
	arTrkBarValueType: ARRAY [0..23] OF UINT; {DE:"Array of value of horizontal bar"}
	arTrkBarName: ARRAY [0..23] OF UDINT; {DE:"Array of names of horizontal bar"}
	arTrkBarCol: ARRAY [0..23] OF UDINT; {DE:"Array of colors of horizontal bar"}
	arTrkMinScale: ARRAY [0..7] OF UDINT; {DE:"Array of min scale y acceptable"}
	arTrkLineWidth: ARRAY [0..7] OF USINT; {DE:"Array of track line widths"}
	rulerXBigMarks: UINT; {DE:"Number of big marks on the X axis"}
	rulerXSmallMarks: UINT; {DE:"Number of small marks on the X axis"}
	rulerYBigMarks: UINT; {DE:"Number of big marks on the Y axis"}
	rulerYSmallMarks: UINT; {DE:"Number of small marks on the Y axis"}
	bEmbeddedXFormat : BOOL; {DE:"Use embedded formats for X labels"}
	bShowAcquisitions : BOOL; {DE:"Show acquisition points on the line"}
	XAxisMode : USINT;   {DE:"X scale mode: 0=scale/offset 1=min/max"}
	arTrkYAxisMode : ARRAY [0..7] OF USINT;   {DE:"Array of track Y scale mode: 0=scale/offset 1=min/max"}
	maxNSamples: UDINT; {DE:"Max number of samples allowed"}
	END_VAR

	VAR
	memVis : BOOL; {DE:"Visibility status"}
	grx1 : UINT; {DE:"X-coordinate of the upper-left corner of the active area"}
	gry1 : UINT; {DE:"Y-coordinate of the upper-left corner of the active area"}
	grx2 : UINT; {DE:"X-coordinate of the lower-right corner of the active area"}
	gry2 : UINT; {DE:"Y-coordinate of the lower-right corner of the active area"}
	pChart : DWORD; {DE:"Address of the chart"}
	lastIdxSamples: UDINT; {DE:" last index of the array of samples "}

	END_VAR

	{CODE:EMBEDDED}

END_FUNCTION_BLOCK

FUNCTION_BLOCK Trend

	VAR_INPUT
	wHnd : UINT; {DE:"Object handle"}
	x1 : UINT; {DE:"X-coordinate of the upper-left corner"}
	y1 : UINT; {DE:"Y-coordinate of the upper-left corner"}
	x2 : UINT; {DE:"X-coordinate of the lower-right corner"}
	y2 : UINT; {DE:"Y-coordinate of the lower-right corner"}
	pFont : UDINT; {DE:"Address of the font"}
	style : USINT; {DE:"Appearence"}
	bordPts : USINT; {DE:"Border thickness"}
	bordCol : UDINT; {DE:"Border color"}
	backCol : UDINT; {DE:"Background color"}
	tyNSamples : UINT; {DE:"Tipe of sampling time"}
	pNSamples :  UDINT; {DE:"Sampling time in seconds"}
	tyXOffset : UINT;  {DE:"Type of X Offset"}
	pXOffset: UDINT; {DE:"X Offset"}
	tyTrackRight : UINT; {DE:"Right label track type"}
	pTrackRight : UDINT; {DE:"Right label track"}
	tyTrackLeft : UINT; {DE:"Left label track type"}
	pTrackLeft : UDINT; {DE:"left label track"}
	formatLeft :  UDINT; {DE:"format of Y label left"}
	formatRight :  UDINT; {DE:"format of Y label right "}
	fGrid : BOOL; {DE:"Flag for grid display"}
	iDivGridX : UINT; {DE:"Horizontal divisions"}
	iDivGridY : UINT; {DE:"Vertical divisions"}
	accMode : USINT; {DE:"Access mode"}
	iXLabelDiv : UINT; {DE:"How many x label"}
	tyXScaleType : UINT; {DE:"X Scale type"}
	pXScale : UDINT; {DE:"X Scale"}
	pClearVar : UDINT; {DE:"Variabile di clear dei dati"}
	pVisVar : UDINT; {DE:"Address of the visibility variable"}
	pRefrVar: UDINT; {DE:"Address of the refresh variable"}
	format :  UDINT; {DE:"format of X labels"}
	XLabelCol : UDINT;{DE:"Color of X label"}
	iDotStep: UINT; {DE:"distance between points of grid"}
	iSampleBuffer: UINT; {DE:" size of sample buffer "}
	arXBars :  ARRAY [0..2] OF UDINT; {DE:"X Bars"}
	arXBarsType : ARRAY [0..2] OF UINT; {DE:"Type of data of X Bars"}
	arXBarsCol: ARRAY [0..2] OF UDINT; {DE:"Bars colors"}
    GridCol : UDINT;	{DE:"Grid color "}
    BorderGridCol : UDINT;	{DE:"Border grid color "}
	arTrkData : ARRAY [0..7] OF UDINT; {DE:"Array of track data addresses"}
	arTrkType : ARRAY [0..7] OF USINT; {DE:"Data type of the associated variable"}
	arTrkCol : ARRAY [0..7] OF UDINT; {DE:"Array of track colors"}
	arTrkScaleY : ARRAY [0..7] OF UDINT;   {DE:"Array of track scale"}
	arTrkScaleYType: ARRAY [0..7] OF UINT; {DE:"Array of track scale type"}
    arTrkOffset: ARRAY [0..7] OF UDINT;    {DE:"Array of track offset"}
	arTrkOffsetType: ARRAY [0..7] OF UINT; {DE:"Array of track offset type"}
	arTrkVis : ARRAY [0..7] OF UDINT; {DE:"Array of track visibility variables"}
	iYLabelDiv: ARRAY [0..7] OF UINT; {DE:"Array of vertical label"}
	arTrkBarValue: ARRAY [0..23] OF UDINT; {DE:"Array of value of horizontal bar"}
	arTrkBarValueType: ARRAY [0..23] OF UINT; {DE:"Array of value of horizontal bar"}
	arTrkBarName: ARRAY [0..23] OF UDINT; {DE:"Array of names of horizontal bar"}
	arTrkBarCol: ARRAY [0..23] OF UDINT; {DE:"Array of colors of horizontal bar"}
	arTrkMinScale: ARRAY [0..23] OF UDINT; {DE:"Array of min scale y acceptable"}
	END_VAR

	VAR
	memVis : BOOL; {DE:"Visibility status"}
	grx1 : UINT; {DE:"X-coordinate of the upper-left corner of the active area"}
	gry1 : UINT; {DE:"Y-coordinate of the upper-left corner of the active area"}
	grx2 : UINT; {DE:"X-coordinate of the lower-right corner of the active area"}
	gry2 : UINT; {DE:"Y-coordinate of the lower-right corner of the active area"}
	pChart : DWORD; {DE:"Address of the chart"}
	firstSamplingTimeS : UDINT; {DE:"First time of sampling in seconds"}
	firstSamplingTimeMS : UINT; {DE:"milliseconds of first time"}
	lastSamplingTimeS: UDINT; {DE:" last time of sampling in seconds "}
	lastSamplingTimeMS: UINT; {DE:" milliseconds of last time "}
	initDraw : BOOL; {DE:"indicate if it's just do the first time of draw "}
	END_VAR

	{CODE:EMBEDDED}

END_FUNCTION_BLOCK

FUNCTION_BLOCK TextBox

	VAR_INPUT
	wHnd : UINT; {DE:"Object handle"}
	x1 : UINT; {DE:"X-coordinate of the upper-left corner"}
	y1 : UINT; {DE:"Y-coordinate of the upper-left corner"}
	x2 : UINT; {DE:"X-coordinate of the lower-right corner"}
	y2 : UINT; {DE:"Y-coordinate of the lower-right corner"}
	pFont : UDINT; {DE:"Address of the font"}
	style : USINT; {DE:"Appearence"}
	foreCol : UDINT; {DE:"Foreground color"}
	bckCol : UDINT; {DE:"Background color"}
	bordPts : USINT; {DE:"Border thickness"}
	bordCol : UDINT; {DE:"Border color"}
	lineNr : BOOL; {DE: "Flag for row number visualization"}
	rw : BOOL; {DE:"Flag of write-mode enabled"}
	pVar : UDINT; {DE:"Address of the associated string"}
	szpVar: UDINT; {DE:"Length of the associated string"}
	pVisVar : UDINT; {DE:"Address of the visibility variable"}
	order : USINT; {DE:"Selection order"}
	accMode : USINT; {DE:"Access mode"}
	rqCursPos: UINT; {DE:"Requested cursor position from the start of the string"}
	rqCursRow: UINT; {DE:"Requested absolute cursor row"}
	dispCurs: BOOL; {DE:"Cursor display flag"}
	dispRow: BOOL; {DE:"Current row selection flag"}
	bckSelCol : UDINT; {DE:"Background selection color"}
	wParam  : UINT;     {DE:"16-bit unsigned parameter"}
	lParam  : DINT;     {DE:"32-bit signed parameter"}
	END_VAR

	VAR_OUTPUT
	outKey : SINT; {DE:"Key pressed to exit the edit mode"}
	outCursPos: UINT; {DE:"Current cursor position from the start of the string"}
	outCursRow: UINT; {DE:"Current absolute cursor row"}
	END_VAR

	VAR
	memVis : BOOL; {DE:"Visibility status"}
	base : UINT; {DE:"Base of the scrolling"}
	END_VAR

	{CODE:EMBEDDED}

END_FUNCTION_BLOCK

FUNCTION_BLOCK CustomCtrl

	VAR_INPUT
	wHnd : UINT; {DE:"Object handle"}
	x1 : UINT; {DE:"X-coordinate of the upper-left corner"}
	y1 : UINT; {DE:"Y-coordinate of the upper-left corner"}
	x2 : UINT; {DE:"X-coordinate of the lower-right corner"}
	y2 : UINT; {DE:"Y-coordinate of the lower-right corner"}
	wCtrlID : UINT; {DE:"Control type"}
	pVisVar : UDINT; {DE:"Address of the visibility flag"}
	refr : BOOL; {DE:"Flag of refresh required"}
	accMode : UINT; {DE:"Access mode"}
	wParam : UINT; {DE:"Unsigned 16-bit input parameter"}
	lParam : DINT; {DE:"Signed 32-bit input parameter"}
	rParam : REAL; {DE:"32-bit real input parameter"}
	END_VAR

	VAR
	memVis : BOOL; {DE:"Visibility status"}
	ptrFunct : UDINT; {DE:"Internal address to the management function"}
	data0 : UDINT; {DE:"Custom control data"}
	data1 : UDINT; {DE:"Custom control data"}
	data2 : UDINT; {DE:"Custom control data"}
	data3 : UDINT; {DE:"Custom control data"}
	END_VAR

	{CODE:EMBEDDED}

END_FUNCTION_BLOCK

FUNCTION_BLOCK Line01
	VAR_INPUT
		x1 : UINT; {DE:"X-coordinate of the upper-left point"}
		y1 : UINT; {DE:"Y-coordinate of the upper-left point"}
		x2 : UINT; {DE:"X-coordinate of the lower-right point"}
		y2 : UINT; {DE:"Y-coordinate of the lower-right point"}
		accMode : USINT; {DE:"Access mode"}
		bordPts : USINT; {DE:"Border thickness"}
		bordCol : UDINT; {DE:"Border color"}
	END_VAR

	{CODE:EMBEDDED}

END_FUNCTION_BLOCK

FUNCTION_BLOCK Rect01
	VAR_INPUT
		x1 : UINT; {DE:"X-coordinate of the upper-left corner"}
		y1 : UINT; {DE:"Y-coordinate of the upper-left corner"}
		x2 : UINT; {DE:"X-coordinate of the lower-right corner"}
		y2 : UINT; {DE:"Y-coordinate of the lower-right corner"}
		accMode : USINT; {DE:"Access mode"}
		transp : USINT; {DE:"Transparent background"}
		bordPts : USINT; {DE:"Border thickness"}
		bordCol : UDINT; {DE:"Border color"}
		bckCol : UDINT; {DE:"Background color"}
	END_VAR

	{CODE:EMBEDDED}

END_FUNCTION_BLOCK
